KUKA KRL program: EPS_2_251806_MH43A_A_20260213065137.src

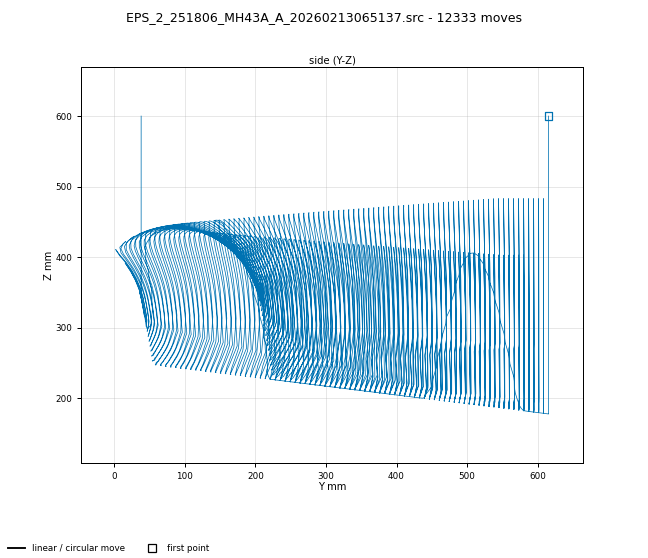
[picture p0: tool path of EPS_2_251806_MH43A_A_20260213065137.src, 12333 of 12335 moves have a stored position in this frame; points joined in program order, loops and branches not executed]
&ACCESS RVP
&REL 4
&COMMENT QRS 19112012
&PARAM EDITMASK = *
DEF PART()
EXT BAS (BAS_COMMAND :IN,REAL :IN )
INT I
BAS (#INITMOV,0 )

;KUKA QRS Post kuka4.cps  Date:22-06-2017 !

File_ID=3028

QRS_PRE_INIT()

;Init var - Until changes are made in qrs_pre_init
Outlet_Square_prg=0
Inlet_1_Square_prg=0
Inlet_2_Square_prg=0
Inlet_3_Square_prg=0
Inlet_4_Square_prg=0
Inlet_5_Square_prg=0

Outlet_1={X 0.000, Y 540.910, Z 382.500, B 0.000, E1 0.000 }
Inlet_1={X 0.000, Y 546.610, Z 302.500, B 0.000, E1 128.000 }
Outlet_1_type=201
Inlet_1_type=201
;QRS#1=Sidecore dimensions
;QRS#2=200-8" PVC SDR 35
;QRS#3=200-8" PVC SDR 35
;QRS#4=
;QRS#5=
;QRS#6=
;QRS#7=
;QRS#8=
;QRS#9=12-08 PSX
;QRS#10=12-08 PSX
;QRS#11=
;QRS#12=
;QRS#13=
;QRS#14=
;QRS#15=
;QRS#16=1220x127x762 2,5'
;QRS#17=EPS Height
;QRS#18=483
;QRS#19=*
;QRS#20= UPDATED VERSION 22-06-2017
;QRS#21=*
Outlet_Square=0100
Inlet_1_Square=0100
Inlet_2_Square=0
Inlet_3_Square=0
Inlet_4_Square=0
Inlet_5_Square=0
Mill_Square=1
Outlet_Square_Prg=204
Inlet_1_Square_prg=204

QRS_INIT()

$ADVANCE=5

; T1
PTP {E1 173.629,E2 173.629}
PTP {X 0,Y 615.469,A -85,B 0,C 180,E1 173.629,E2 173.629,E3 0,E4 0,E5 0,E6 0}
QRS_SPEED_INIT()
LIN {X 0,Y 615.469,Z 600,A -85,B 0,C 180,E1 173.629,E2 173.629,E3 0,E4 0,E5 0,E6 0} C_VEL
LIN {X 0,Y 615.469,Z 187.869,A -85,B 0,C 180,E1 173.629,E2 173.629} C_VEL
LIN {X 0,Y 615.469,Z 179.692,A -85,B 0,C 180,E1 173.629,E2 173.629} C_VEL
LIN {X 0,Y 615.462,Z 177.692,A -85,B 0,C 180,E1 173.442,E2 173.442} C_VEL
LIN {X 0,Y 615.491,Z 177.698,A -85,B 0,C 180,E1 170.801,E2 170.801} C_VEL
LIN {X 0,Y 615.483,Z 177.684,A -85,B 0,C 180,E1 168.139,E2 168.139} C_VEL
LIN {X 0,Y 615.47,Z 177.694,A -85,B 0,C 180,E1 165.451,E2 165.451} C_VEL
LIN {X 0,Y 615.488,Z 177.69,A -85,B 0,C 180,E1 162.73,E2 162.73} C_VEL
LIN {X 0,Y 615.467,Z 177.689,A -85,B 0,C 180,E1 159.967,E2 159.967} C_VEL
LIN {X 0,Y 615.467,Z 177.789,A -85,B 0,C 180,E1 157.786,E2 157.786} C_VEL
LIN {X 0,Y 615.492,Z 192.068,A -85,B 0,C 180,E1 155.008,E2 155.008} C_VEL
LIN {X 0,Y 615.496,Z 193.094,A -85,B 0,C 180,E1 154.81,E2 154.81} C_VEL
LIN {X 0,Y 615.476,Z 299.263,A -85,B 0,C 180,E1 153.537,E2 153.537} C_VEL
LIN {X 0,Y 615.469,Z 311.971,A -85,B 0,C 180,E1 153.256,E2 153.256} C_VEL
LIN {X 0,Y 615.481,Z 325.146,A -85,B 0,C 180,E1 152.822,E2 152.822} C_VEL
LIN {X 0,Y 615.472,Z 337.362,A -85,B 0,C 180,E1 152.269,E2 152.269} C_VEL
LIN {X 0,Y 615.477,Z 348.518,A -85,B 0,C 180,E1 151.617,E2 151.617} C_VEL
LIN {X 0,Y 615.5,Z 358.718,A -85,B 0,C 180,E1 150.876,E2 150.876} C_VEL
LIN {X 0,Y 615.498,Z 368.216,A -85,B 0,C 180,E1 150.022,E2 150.022} C_VEL
LIN {X 0,Y 615.497,Z 376.701,A -85,B 0,C 180,E1 149.081,E2 149.081} C_VEL
LIN {X 0,Y 615.498,Z 383.508,A -85,B 0,C 180,E1 148.154,E2 148.154} C_VEL
LIN {X 0,Y 615.495,Z 389.434,A -85,B 0,C 180,E1 147.154,E2 147.154} C_VEL
LIN {X 0,Y 615.495,Z 394.787,A -85,B 0,C 180,E1 145.978,E2 145.978} C_VEL
LIN {X 0,Y 615.497,Z 398.663,A -85,B 0,C 180,E1 144.786,E2 144.786} C_VEL
LIN {X 0,Y 615.494,Z 401.179,A -85,B 0,C 180,E1 143.576,E2 143.576} C_VEL
LIN {X 0,Y 615.496,Z 402.068,A -85,B 0,C 180,E1 142.758,E2 142.758} C_VEL
LIN {X 0,Y 615.494,Z 402.388,A -85,B 0,C 180,E1 141.932,E2 141.932} C_VEL
LIN {X 0,Y 615.495,Z 401.914,A -85,B 0,C 180,E1 140.937,E2 140.937} C_VEL
LIN {X 0,Y 615.496,Z 400.471,A -85,B 0,C 180,E1 139.91,E2 139.91} C_VEL
LIN {X 0,Y 615.494,Z 398.077,A -85,B 0,C 180,E1 138.905,E2 138.905} C_VEL
LIN {X 0,Y 615.497,Z 394.739,A -85,B 0,C 180,E1 137.919,E2 137.919} C_VEL
LIN {X 0,Y 615.498,Z 389.436,A -85,B 0,C 180,E1 136.756,E2 136.756} C_VEL
LIN {X 0,Y 615.494,Z 382.831,A -85,B 0,C 180,E1 135.656,E2 135.656} C_VEL
LIN {X 0,Y 615.495,Z 375.933,A -85,B 0,C 180,E1 134.735,E2 134.735} C_VEL
LIN {X 0,Y 615.498,Z 367.432,A -85,B 0,C 180,E1 133.808,E2 133.808} C_VEL
LIN {X 0,Y 615.499,Z 357.776,A -85,B 0,C 180,E1 132.961,E2 132.961} C_VEL
LIN {X 0,Y 615.47,Z 347.339,A -85,B 0,C 180,E1 132.216,E2 132.216} C_VEL
LIN {X 0,Y 615.466,Z 337.073,A -85,B 0,C 180,E1 131.625,E2 131.625} C_VEL
LIN {X 0,Y 615.489,Z 325.328,A -85,B 0,C 180,E1 131.094,E2 131.094} C_VEL
LIN {X 0,Y 615.476,Z 312.489,A -85,B 0,C 180,E1 130.668,E2 130.668} C_VEL
LIN {X 0,Y 615.478,Z 299.674,A -85,B 0,C 180,E1 130.381,E2 130.381} C_VEL
LIN {X 0,Y 615.5,Z 193.126,A -85,B 0,C 180,E1 129.106,E2 129.106} C_VEL
LIN {X 0,Y 615.473,Z 179.33,A -85,B 0,C 180,E1 126.426,E2 126.426} C_VEL
LIN {X 0,Y 615.455,Z 177.694,A -85,B 0,C 180,E1 126.09,E2 126.09} C_VEL
LIN {X 0,Y 615.472,Z 177.687,A -85,B 0,C 180,E1 123.532,E2 123.532} C_VEL
LIN {X 0,Y 615.494,Z 177.696,A -85,B 0,C 180,E1 120.919,E2 120.919} C_VEL
LIN {X 0,Y 615.464,Z 177.696,A -85,B 0,C 180,E1 118.446,E2 118.446} C_VEL
LIN {X 0,Y 615.461,Z 177.695,A -85,B 0,C 180,E1 116.445,E2 116.445} C_VEL
LIN {X 0,Y 615.456,Z 177.69,A -85,B 0,C 180,E1 114.001,E2 114.001} C_VEL
LIN {X 0,Y 615.496,Z 177.687,A -85,B 0,C 180,E1 111.431,E2 111.431} C_VEL
LIN {X 0,Y 615.459,Z 177.695,A -85,B 0,C 180,E1 108.596,E2 108.596} C_VEL
LIN {X 0,Y 615.472,Z 177.687,A -85,B 0,C 180,E1 105.905,E2 105.905} C_VEL
LIN {X 0,Y 615.495,Z 177.701,A -85,B 0,C 180,E1 103.201,E2 103.201} C_VEL
LIN {X 0,Y 615.451,Z 177.693,A -85,B 0,C 180,E1 100.527,E2 100.527} C_VEL
LIN {X 0,Y 615.484,Z 177.687,A -85,B 0,C 180,E1 97.875,E2 97.875} C_VEL
LIN {X 0,Y 615.485,Z 177.699,A -85,B 0,C 180,E1 95.241,E2 95.241} C_VEL
LIN {X 0,Y 615.451,Z 177.692,A -85,B 0,C 180,E1 92.618,E2 92.618} C_VEL
LIN {X 0,Y 615.486,Z 177.688,A -85,B 0,C 180,E1 90,E2 90} C_VEL
LIN {X 0,Y 615.48,Z 177.698,A -85,B 0,C 180,E1 87.382,E2 87.382} C_VEL
LIN {X 0,Y 615.447,Z 177.692,A -85,B 0,C 180,E1 84.758,E2 84.758} C_VEL
LIN {X 0,Y 615.489,Z 177.689,A -85,B 0,C 180,E1 82.124,E2 82.124} C_VEL
LIN {X 0,Y 615.47,Z 177.697,A -85,B 0,C 180,E1 79.473,E2 79.473} C_VEL
LIN {X 0,Y 615.455,Z 177.69,A -85,B 0,C 180,E1 76.798,E2 76.798} C_VEL
LIN {X 0,Y 615.495,Z 177.693,A -85,B 0,C 180,E1 74.095,E2 74.095} C_VEL
LIN {X 0,Y 615.451,Z 177.694,A -85,B 0,C 180,E1 71.353,E2 71.353} C_VEL
LIN {X 0,Y 615.448,Z 177.693,A -85,B 0,C 180,E1 69.268,E2 69.268} C_VEL
LIN {X 0,Y 615.488,Z 177.69,A -85,B 0,C 180,E1 66.443,E2 66.443} C_VEL
LIN {X 0,Y 615.45,Z 177.695,A -85,B 0,C 180,E1 63.554,E2 63.554} C_VEL
LIN {X 0,Y 615.448,Z 177.692,A -85,B 0,C 180,E1 61.34,E2 61.34} C_VEL
LIN {X 0,Y 615.474,Z 177.688,A -85,B 0,C 180,E1 58.916,E2 58.916} C_VEL
LIN {X 0,Y 615.465,Z 177.697,A -85,B 0,C 180,E1 55.976,E2 55.976} C_VEL
LIN {X 0,Y 615.445,Z 177.693,A -85,B 0,C 180,E1 53.572,E2 53.572} C_VEL
LIN {X 0,Y 615.491,Z 177.687,A -85,B 0,C 180,E1 50.938,E2 50.938} C_VEL
LIN {X 0,Y 615.495,Z 177.7,A -85,B 0,C 180,E1 48.526,E2 48.526} C_VEL
LIN {X 0,Y 615.446,Z 177.694,A -85,B 0,C 180,E1 45.846,E2 45.846} C_VEL
LIN {X 0,Y 615.488,Z 177.689,A -85,B 0,C 180,E1 43.047,E2 43.047} C_VEL
LIN {X 0,Y 615.481,Z 177.702,A -85,B 0,C 180,E1 40.607,E2 40.607} C_VEL
LIN {X 0,Y 615.444,Z 177.694,A -85,B 0,C 180,E1 38.006,E2 38.006} C_VEL
LIN {X 0,Y 615.454,Z 177.691,A -85,B 0,C 180,E1 35.618,E2 35.618} C_VEL
LIN {X 0,Y 615.488,Z 177.69,A -85,B 0,C 180,E1 33.236,E2 33.236} C_VEL
LIN {X 0,Y 615.493,Z 177.701,A -85,B 0,C 180,E1 30.919,E2 30.919} C_VEL
LIN {X 0,Y 615.451,Z 177.696,A -85,B 0,C 180,E1 28.443,E2 28.443} C_VEL
LIN {X 0,Y 615.449,Z 177.695,A -85,B 0,C 180,E1 26.446,E2 26.446} C_VEL
LIN {X 0,Y 615.449,Z 177.692,A -85,B 0,C 180,E1 23.999,E2 23.999} C_VEL
LIN {X 0,Y 615.497,Z 177.69,A -85,B 0,C 180,E1 21.432,E2 21.432} C_VEL
LIN {X 0,Y 615.444,Z 177.696,A -85,B 0,C 180,E1 18.592,E2 18.592} C_VEL
LIN {X 0,Y 615.443,Z 177.694,A -85,B 0,C 180,E1 16.416,E2 16.416} C_VEL
LIN {X 0,Y 615.477,Z 177.689,A -85,B 0,C 180,E1 13.874,E2 13.874} C_VEL
LIN {X 0,Y 615.476,Z 177.699,A -85,B 0,C 180,E1 11.193,E2 11.193} C_VEL
LIN {X 0,Y 615.442,Z 177.693,A -85,B 0,C 180,E1 8.537,E2 8.537} C_VEL
LIN {X 0,Y 615.496,Z 177.688,A -85,B 0,C 180,E1 5.898,E2 5.898} C_VEL
LIN {X 0,Y 615.466,Z 177.698,A -85,B 0,C 180,E1 3.273,E2 3.273} C_VEL
LIN {X 0,Y 615.465,Z 177.698,A -85,B 0,C 180,E1 1.309,E2 1.309} C_VEL
LIN {X 0,Y 615.442,Z 177.693,A -85,B 0,C 180,E1 -1.309,E2 -1.309} C_VEL
LIN {X 0,Y 615.487,Z 177.692,A -85,B 0,C 180,E1 -3.929,E2 -3.929} C_VEL
LIN {X 0,Y 615.456,Z 177.698,A -85,B 0,C 180,E1 -6.557,E2 -6.557} C_VEL
LIN {X 0,Y 615.458,Z 177.697,A -85,B 0,C 180,E1 -8.537,E2 -8.537} C_VEL
LIN {X 0,Y 615.44,Z 177.695,A -85,B 0,C 180,E1 -10.863,E2 -10.863} C_VEL
LIN {X 0,Y 615.449,Z 177.692,A -85,B 0,C 180,E1 -13.202,E2 -13.202} C_VEL
LIN {X 0,Y 615.493,Z 177.699,A -85,B 0,C 180,E1 -15.905,E2 -15.905} C_VEL
LIN {X 0,Y 615.438,Z 177.696,A -85,B 0,C 180,E1 -18.648,E2 -18.648} C_VEL
LIN {X 0,Y 615.488,Z 177.689,A -85,B 0,C 180,E1 -21.432,E2 -21.432} C_VEL
LIN {X 0,Y 615.449,Z 177.697,A -85,B 0,C 180,E1 -24.274,E2 -24.274} C_VEL
LIN {X 0,Y 615.438,Z 177.696,A -85,B 0,C 180,E1 -26.447,E2 -26.447} C_VEL
LIN {X 0,Y 615.439,Z 177.694,A -85,B 0,C 180,E1 -28.661,E2 -28.661} C_VEL
LIN {X 0,Y 615.471,Z 177.691,A -85,B 0,C 180,E1 -31.083,E2 -31.083} C_VEL
LIN {X 0,Y 615.449,Z 177.697,A -85,B 0,C 180,E1 -34.025,E2 -34.025} C_VEL
LIN {X 0,Y 615.437,Z 177.694,A -85,B 0,C 180,E1 -36.428,E2 -36.428} C_VEL
LIN {X 0,Y 615.49,Z 177.69,A -85,B 0,C 180,E1 -39.062,E2 -39.062} C_VEL
LIN {X 0,Y 615.487,Z 177.699,A -85,B 0,C 180,E1 -41.474,E2 -41.474} C_VEL
LIN {X 0,Y 615.435,Z 177.695,A -85,B 0,C 180,E1 -44.155,E2 -44.155} C_VEL
LIN {X 0,Y 615.473,Z 177.691,A -85,B 0,C 180,E1 -46.754,E2 -46.754} C_VEL
LIN {X 0,Y 615.469,Z 177.7,A -85,B 0,C 180,E1 -49.392,E2 -49.392} C_VEL
LIN {X 0,Y 615.434,Z 177.696,A -85,B 0,C 180,E1 -51.927,E2 -51.927} C_VEL
LIN {X 0,Y 615.449,Z 177.693,A -85,B 0,C 180,E1 -54.381,E2 -54.381} C_VEL
LIN {X 0,Y 615.489,Z 177.694,A -85,B 0,C 180,E1 -56.764,E2 -56.764} C_VEL
LIN {X 0,Y 615.477,Z 177.701,A -85,B 0,C 180,E1 -59.079,E2 -59.079} C_VEL
LIN {X 0,Y 615.437,Z 177.697,A -85,B 0,C 180,E1 -61.559,E2 -61.559} C_VEL
LIN {X 0,Y 615.436,Z 177.696,A -85,B 0,C 180,E1 -63.553,E2 -63.553} C_VEL
LIN {X 0,Y 615.445,Z 177.839,A -85,B 0,C 180,E1 -66.029,E2 -66.029} C_VEL
LIN {X 0,Y 615.472,Z 199.807,A -85,B 0,C 180,E1 -68.743,E2 -68.743} C_VEL
LIN {X 0,Y 615.494,Z 221.654,A -85,B 0,C 180,E1 -71.394,E2 -71.394} C_VEL
LIN {X 0,Y 615.491,Z 245.672,A -85,B 0,C 180,E1 -74.265,E2 -74.265} C_VEL
LIN {X 0,Y 615.455,Z 269.639,A -85,B 0,C 180,E1 -77.092,E2 -77.092} C_VEL
LIN {X 0,Y 615.457,Z 274.667,A -85,B 0,C 180,E1 -77.176,E2 -77.176} C_VEL
LIN {X 0,Y 615.488,Z 378.818,A -85,B 0,C 180,E1 -78.41,E2 -78.41} C_VEL
LIN {X 0,Y 615.477,Z 391.338,A -85,B 0,C 180,E1 -78.681,E2 -78.681} C_VEL
LIN {X 0,Y 615.488,Z 404.617,A -85,B 0,C 180,E1 -79.113,E2 -79.113} C_VEL
LIN {X 0,Y 615.477,Z 416.475,A -85,B 0,C 180,E1 -79.639,E2 -79.639} C_VEL
LIN {X 0,Y 615.494,Z 427.991,A -85,B 0,C 180,E1 -80.304,E2 -80.304} C_VEL
LIN {X 0,Y 615.499,Z 438.338,A -85,B 0,C 180,E1 -81.05,E2 -81.05} C_VEL
LIN {X 0,Y 615.497,Z 446.809,A -85,B 0,C 180,E1 -81.794,E2 -81.794} C_VEL
LIN {X 0,Y 615.498,Z 454.604,A -85,B 0,C 180,E1 -82.619,E2 -82.619} C_VEL
LIN {X 0,Y 615.496,Z 462.202,A -85,B 0,C 180,E1 -83.608,E2 -83.608} C_VEL
LIN {X 0,Y 615.498,Z 469.203,A -85,B 0,C 180,E1 -84.759,E2 -84.759} C_VEL
LIN {X 0,Y 615.494,Z 473.85,A -85,B 0,C 180,E1 -85.743,E2 -85.743} C_VEL
LIN {X 0,Y 615.494,Z 477.398,A -85,B 0,C 180,E1 -86.727,E2 -86.727} C_VEL
LIN {X 0,Y 615.497,Z 479.232,A -85,B 0,C 180,E1 -87.382,E2 -87.382} C_VEL
LIN {X 0,Y 615.5,Z 480.607,A -85,B 0,C 180,E1 -88.037,E2 -88.037} C_VEL
LIN {X 0,Y 615.496,Z 482.173,A -85,B 0,C 180,E1 -89.346,E2 -89.346} C_VEL
LIN {X 0,Y 615.494,Z 482.389,A -85,B 0,C 180,E1 -90,E2 -90} C_VEL
LIN {X 0,Y 615.495,Z 481.58,A -85,B 0,C 180,E1 -91.308,E2 -91.308} C_VEL
LIN {X 0,Y 615.5,Z 480.608,A -85,B 0,C 180,E1 -91.963,E2 -91.963} C_VEL
LIN {X 0,Y 615.497,Z 479.233,A -85,B 0,C 180,E1 -92.618,E2 -92.618} C_VEL
LIN {X 0,Y 615.496,Z 476.35,A -85,B 0,C 180,E1 -93.6,E2 -93.6} C_VEL
LIN {X 0,Y 615.498,Z 472.442,A -85,B 0,C 180,E1 -94.584,E2 -94.584} C_VEL
LIN {X 0,Y 615.499,Z 467.406,A -85,B 0,C 180,E1 -95.57,E2 -95.57} C_VEL
LIN {X 0,Y 615.497,Z 460.87,A -85,B 0,C 180,E1 -96.583,E2 -96.583} C_VEL
LIN {X 0,Y 615.497,Z 453.134,A -85,B 0,C 180,E1 -97.545,E2 -97.545} C_VEL
LIN {X 0,Y 615.498,Z 445.047,A -85,B 0,C 180,E1 -98.371,E2 -98.371} C_VEL
LIN {X 0,Y 615.499,Z 435.169,A -85,B 0,C 180,E1 -99.198,E2 -99.198} C_VEL
LIN {X 0,Y 615.488,Z 423.984,A -85,B 0,C 180,E1 -99.945,E2 -99.945} C_VEL
LIN {X 0,Y 615.482,Z 413.027,A -85,B 0,C 180,E1 -100.527,E2 -100.527} C_VEL
LIN {X 0,Y 615.48,Z 400.492,A -85,B 0,C 180,E1 -101.04,E2 -101.04} C_VEL
LIN {X 0,Y 615.479,Z 388.073,A -85,B 0,C 180,E1 -101.402,E2 -101.402} C_VEL
LIN {X 0,Y 615.493,Z 374.475,A -85,B 0,C 180,E1 -101.652,E2 -101.652} C_VEL
LIN {X 0,Y 615.455,Z 269.821,A -85,B 0,C 180,E1 -102.887,E2 -102.887} C_VEL
LIN {X 0,Y 615.493,Z 247.108,A -85,B 0,C 180,E1 -105.565,E2 -105.565} C_VEL
LIN {X 0,Y 615.49,Z 223.006,A -85,B 0,C 180,E1 -108.443,E2 -108.443} C_VEL
LIN {X 0,Y 615.46,Z 201.245,A -85,B 0,C 180,E1 -111.082,E2 -111.082} C_VEL
LIN {X 0,Y 615.447,Z 178.059,A -85,B 0,C 180,E1 -113.943,E2 -113.943} C_VEL
LIN {X 0,Y 615.443,Z 177.694,A -85,B 0,C 180,E1 -113.999,E2 -113.999} C_VEL
LIN {X 0,Y 615.437,Z 177.696,A -85,B 0,C 180,E1 -116.446,E2 -116.446} C_VEL
LIN {X 0,Y 615.485,Z 177.692,A -85,B 0,C 180,E1 -119.406,E2 -119.406} C_VEL
LIN {X 0,Y 615.455,Z 177.692,A -85,B 0,C 180,E1 -121.687,E2 -121.687} C_VEL
LIN {X 0,Y 615.438,Z 177.694,A -85,B 0,C 180,E1 -124.025,E2 -124.025} C_VEL
LIN {X 0,Y 615.489,Z 177.699,A -85,B 0,C 180,E1 -126.936,E2 -126.936} C_VEL
LIN {X 0,Y 615.441,Z 177.693,A -85,B 0,C 180,E1 -129.754,E2 -129.754} C_VEL
LIN {X 0,Y 615.462,Z 177.698,A -85,B 0,C 180,E1 -132.355,E2 -132.355} C_VEL
LIN {X 0,Y 615.491,Z 177.688,A -85,B 0,C 180,E1 -135.068,E2 -135.068} C_VEL
LIN {X 0,Y 615.444,Z 177.693,A -85,B 0,C 180,E1 -137.643,E2 -137.643} C_VEL
LIN {X 0,Y 615.474,Z 177.698,A -85,B 0,C 180,E1 -140.249,E2 -140.249} C_VEL
LIN {X 0,Y 615.471,Z 177.689,A -85,B 0,C 180,E1 -143.065,E2 -143.065} C_VEL
LIN {X 0,Y 615.452,Z 177.691,A -85,B 0,C 180,E1 -145.304,E2 -145.304} C_VEL
LIN {X 0,Y 615.451,Z 177.695,A -85,B 0,C 180,E1 -147.675,E2 -147.675} C_VEL
LIN {X 0,Y 615.499,Z 177.7,A -85,B 0,C 180,E1 -150.203,E2 -150.203} C_VEL
LIN {X 0,Y 615.462,Z 177.689,A -85,B 0,C 180,E1 -152.96,E2 -152.96} C_VEL
LIN {X 0,Y 615.458,Z 177.69,A -85,B 0,C 180,E1 -155.007,E2 -155.007} C_VEL
LIN {X 0,Y 615.467,Z 177.697,A -85,B 0,C 180,E1 -157.659,E2 -157.659} C_VEL
LIN {X 0,Y 615.475,Z 177.687,A -85,B 0,C 180,E1 -160.662,E2 -160.662} C_VEL
LIN {X 0,Y 615.466,Z 177.688,A -85,B 0,C 180,E1 -162.729,E2 -162.729} C_VEL
LIN {X 0,Y 615.469,Z 177.697,A -85,B 0,C 180,E1 -165.45,E2 -165.45} C_VEL
LIN {X 0,Y 615.488,Z 177.689,A -85,B 0,C 180,E1 -168.139,E2 -168.139} C_VEL
LIN {X 0,Y 615.457,Z 177.69,A -85,B 0,C 180,E1 -170.801,E2 -170.801} C_VEL
LIN {X 0,Y 615.49,Z 177.699,A -85,B 0,C 180,E1 -173.443,E2 -173.443} C_VEL
LIN {X 0,Y 615.487,Z 177.686,A -85,B 0,C 180,E1 -176.071,E2 -176.071} C_VEL
LIN {X 0,Y 615.459,Z 177.691,A -85,B 0,C 180,E1 -178.691,E2 -178.691} C_VEL
LIN {X 0,Y 615.492,Z 177.702,A -85,B 0,C 180,E1 -181.309,E2 -181.309} C_VEL
LIN {X 0,Y 615.486,Z 177.685,A -85,B 0,C 180,E1 -183.928,E2 -183.928} C_VEL
LIN {X 0,Y 615.462,Z 177.692,A -85,B 0,C 180,E1 -186.558,E2 -186.558} C_VEL
LIN {X 0,Y 614.804,Z 177.845,A -85,B 0,C 180,E1 -187.104,E2 -187.104} C_VEL
LIN {X 0,Y 611.985,Z 178.248,A -85,B 0,C 180,E1 -187.99,E2 -187.99} C_VEL
LIN {X 0,Y 609.595,Z 178.562,A -85,B 0,C 180,E1 -188.703,E2 -188.703} C_VEL
LIN {X 0,Y 608.556,Z 178.683,A -85,B 0,C 180,E1 -189.252,E2 -189.252} C_VEL
LIN {X 0,Y 608.464,Z 178.691,A -85,B 0,C 180,E1 -189.438,E2 -189.438} C_VEL
LIN {X 0,Y 608.456,Z 178.687,A -85,B 0,C 180,E1 -192,E2 -192} C_VEL
LIN {X 0,Y 608.466,Z 178.693,A -85,B 0,C 180,E1 -194.721,E2 -194.721} C_VEL
LIN {X 0,Y 608.45,Z 178.69,A -85,B 0,C 180,E1 -197.477,E2 -197.477} C_VEL
LIN {X 0,Y 608.449,Z 178.691,A -85,B 0,C 180,E1 -200.275,E2 -200.275} C_VEL
LIN {X 0,Y 608.454,Z 178.73,A -85,B 0,C 180,E1 -202.183,E2 -202.183} C_VEL
LIN {X 0,Y 608.474,Z 192.782,A -85,B 0,C 180,E1 -204.935,E2 -204.935} C_VEL
LIN {X 0,Y 608.458,Z 193.373,A -85,B 0,C 180,E1 -205.049,E2 -205.049} C_VEL
LIN {X 0,Y 608.535,Z 299.465,A -85,B 0,C 180,E1 -206.331,E2 -206.331} C_VEL
LIN {X 0,Y 608.52,Z 312.77,A -85,B 0,C 180,E1 -206.632,E2 -206.632} C_VEL
LIN {X 0,Y 608.504,Z 323.878,A -85,B 0,C 180,E1 -206.999,E2 -206.999} C_VEL
LIN {X 0,Y 608.502,Z 335.659,A -85,B 0,C 180,E1 -207.515,E2 -207.515} C_VEL
LIN {X 0,Y 608.458,Z 347.236,A -85,B 0,C 180,E1 -208.173,E2 -208.173} C_VEL
LIN {X 0,Y 608.486,Z 357.461,A -85,B 0,C 180,E1 -208.901,E2 -208.901} C_VEL
LIN {X 0,Y 608.483,Z 367.48,A -85,B 0,C 180,E1 -209.779,E2 -209.779} C_VEL
LIN {X 0,Y 608.459,Z 376.171,A -85,B 0,C 180,E1 -210.726,E2 -210.726} C_VEL
LIN {X 0,Y 608.463,Z 383.466,A -85,B 0,C 180,E1 -211.705,E2 -211.705} C_VEL
LIN {X 0,Y 608.432,Z 388.454,A -85,B 0,C 180,E1 -212.518,E2 -212.518} C_VEL
LIN {X 0,Y 608.425,Z 394.325,A -85,B 0,C 180,E1 -213.728,E2 -213.728} C_VEL
LIN {X 0,Y 608.427,Z 398.485,A -85,B 0,C 180,E1 -214.903,E2 -214.903} C_VEL
LIN {X 0,Y 608.422,Z 401.259,A -85,B 0,C 180,E1 -216.094,E2 -216.094} C_VEL
LIN {X 0,Y 608.435,Z 402.622,A -85,B 0,C 180,E1 -217.154,E2 -217.154} C_VEL
LIN {X 0,Y 608.42,Z 402.962,A -85,B 0,C 180,E1 -218.235,E2 -218.235} C_VEL
LIN {X 0,Y 608.423,Z 402.096,A -85,B 0,C 180,E1 -219.443,E2 -219.443} C_VEL
LIN {X 0,Y 608.433,Z 399.686,A -85,B 0,C 180,E1 -220.74,E2 -220.74} C_VEL
LIN {X 0,Y 608.45,Z 396.943,A -85,B 0,C 180,E1 -221.673,E2 -221.673} C_VEL
LIN {X 0,Y 608.442,Z 393.221,A -85,B 0,C 180,E1 -222.62,E2 -222.62} C_VEL
LIN {X 0,Y 608.453,Z 388.509,A -85,B 0,C 180,E1 -223.562,E2 -223.562} C_VEL
LIN {X 0,Y 608.459,Z 381.684,A -85,B 0,C 180,E1 -224.648,E2 -224.648} C_VEL
LIN {X 0,Y 608.469,Z 372.97,A -85,B 0,C 180,E1 -225.735,E2 -225.735} C_VEL
LIN {X 0,Y 608.476,Z 364.473,A -85,B 0,C 180,E1 -226.595,E2 -226.595} C_VEL
LIN {X 0,Y 608.478,Z 354.93,A -85,B 0,C 180,E1 -227.386,E2 -227.386} C_VEL
LIN {X 0,Y 608.475,Z 343.681,A -85,B 0,C 180,E1 -228.135,E2 -228.135} C_VEL
LIN {X 0,Y 608.512,Z 331.514,A -85,B 0,C 180,E1 -228.774,E2 -228.774} C_VEL
LIN {X 0,Y 608.526,Z 318.947,A -85,B 0,C 180,E1 -229.268,E2 -229.268} C_VEL
LIN {X 0,Y 608.518,Z 305.883,A -85,B 0,C 180,E1 -229.632,E2 -229.632} C_VEL
LIN {X 0,Y 608.543,Z 293.08,A -85,B 0,C 180,E1 -229.853,E2 -229.853} C_VEL
LIN {X 0,Y 608.5,Z 193.71,A -85,B 0,C 180,E1 -231.03,E2 -231.03} C_VEL
LIN {X 0,Y 608.473,Z 193.319,A -85,B 0,C 180,E1 -231.051,E2 -231.051} C_VEL
LIN {X 0,Y 608.458,Z 179.763,A -85,B 0,C 180,E1 -233.704,E2 -233.704} C_VEL
LIN {X 0,Y 608.437,Z 178.692,A -85,B 0,C 180,E1 -233.956,E2 -233.956} C_VEL
LIN {X 0,Y 608.443,Z 178.689,A -85,B 0,C 180,E1 -236.328,E2 -236.328} C_VEL
LIN {X 0,Y 608.449,Z 178.691,A -85,B 0,C 180,E1 -238.732,E2 -238.732} C_VEL
LIN {X 0,Y 608.463,Z 178.693,A -85,B 0,C 180,E1 -241.382,E2 -241.382} C_VEL
LIN {X 0,Y 608.427,Z 178.691,A -85,B 0,C 180,E1 -243.964,E2 -243.964} C_VEL
LIN {X 0,Y 608.447,Z 178.688,A -85,B 0,C 180,E1 -246.154,E2 -246.154} C_VEL
LIN {X 0,Y 608.453,Z 178.698,A -85,B 0,C 180,E1 -249.019,E2 -249.019} C_VEL
LIN {X 0,Y 608.426,Z 178.691,A -85,B 0,C 180,E1 -251.828,E2 -251.828} C_VEL
LIN {X 0,Y 608.474,Z 178.691,A -85,B 0,C 180,E1 -254.594,E2 -254.594} C_VEL
LIN {X 0,Y 608.453,Z 178.69,A -85,B 0,C 180,E1 -257.323,E2 -257.323} C_VEL
LIN {X 0,Y 608.453,Z 178.688,A -85,B 0,C 180,E1 -260.023,E2 -260.023} C_VEL
LIN {X 0,Y 608.461,Z 178.697,A -85,B 0,C 180,E1 -262.701,E2 -262.701} C_VEL
LIN {X 0,Y 608.465,Z 178.695,A -85,B 0,C 180,E1 -264.698,E2 -264.698} C_VEL
LIN {X 0,Y 608.447,Z 178.689,A -85,B 0,C 180,E1 -267.352,E2 -267.352} C_VEL
LIN {X 0,Y 608.477,Z 178.687,A -85,B 0,C 180,E1 -270,E2 -270} C_VEL
LIN {X 0,Y 608.47,Z 178.692,A -85,B 0,C 180,E1 -272.648,E2 -272.648} C_VEL
LIN {X 0,Y 608.433,Z 178.69,A -85,B 0,C 180,E1 -275.302,E2 -275.302} C_VEL
LIN {X 0,Y 608.478,Z 178.689,A -85,B 0,C 180,E1 -277.967,E2 -277.967} C_VEL
LIN {X 0,Y 608.443,Z 178.693,A -85,B 0,C 180,E1 -280.65,E2 -280.65} C_VEL
LIN {X 0,Y 608.444,Z 178.689,A -85,B 0,C 180,E1 -283.357,E2 -283.357} C_VEL
LIN {X 0,Y 608.459,Z 178.697,A -85,B 0,C 180,E1 -286.094,E2 -286.094} C_VEL
LIN {X 0,Y 608.44,Z 178.689,A -85,B 0,C 180,E1 -288.87,E2 -288.87} C_VEL
LIN {X 0,Y 608.469,Z 178.691,A -85,B 0,C 180,E1 -291.692,E2 -291.692} C_VEL
LIN {X 0,Y 608.432,Z 178.691,A -85,B 0,C 180,E1 -294.572,E2 -294.572} C_VEL
LIN {X 0,Y 608.466,Z 178.687,A -85,B 0,C 180,E1 -297.205,E2 -297.205} C_VEL
LIN {X 0,Y 608.45,Z 178.695,A -85,B 0,C 180,E1 -299.968,E2 -299.968} C_VEL
LIN {X 0,Y 608.444,Z 178.689,A -85,B 0,C 180,E1 -302.881,E2 -302.881} C_VEL
LIN {X 0,Y 608.44,Z 178.693,A -85,B 0,C 180,E1 -305.278,E2 -305.278} C_VEL
LIN {X 0,Y 608.456,Z 178.695,A -85,B 0,C 180,E1 -307.748,E2 -307.748} C_VEL
LIN {X 0,Y 608.435,Z 178.69,A -85,B 0,C 180,E1 -310.327,E2 -310.327} C_VEL
LIN {X 0,Y 608.449,Z 178.69,A -85,B 0,C 180,E1 -312.961,E2 -312.961} C_VEL
LIN {X 0,Y 608.433,Z 178.695,A -85,B 0,C 180,E1 -315.739,E2 -315.739} C_VEL
LIN {X 0,Y 608.433,Z 178.692,A -85,B 0,C 180,E1 -317.936,E2 -317.936} C_VEL
LIN {X 0,Y 608.442,Z 178.691,A -85,B 0,C 180,E1 -320.706,E2 -320.706} C_VEL
LIN {X 0,Y 608.457,Z 178.695,A -85,B 0,C 180,E1 -323.085,E2 -323.085} C_VEL
LIN {X 0,Y 608.458,Z 178.691,A -85,B 0,C 180,E1 -325.53,E2 -325.53} C_VEL
LIN {X 0,Y 608.436,Z 178.69,A -85,B 0,C 180,E1 -327.904,E2 -327.904} C_VEL
LIN {X 0,Y 608.441,Z 178.689,A -85,B 0,C 180,E1 -330.219,E2 -330.219} C_VEL
LIN {X 0,Y 608.488,Z 178.69,A -85,B 0,C 180,E1 -332.792,E2 -332.792} C_VEL
LIN {X 0,Y 608.435,Z 178.693,A -85,B 0,C 180,E1 -335.428,E2 -335.428} C_VEL
LIN {X 0,Y 608.461,Z 178.688,A -85,B 0,C 180,E1 -338.308,E2 -338.308} C_VEL
LIN {X 0,Y 608.426,Z 178.694,A -85,B 0,C 180,E1 -341.297,E2 -341.297} C_VEL
LIN {X 0,Y 608.436,Z 178.69,A -85,B 0,C 180,E1 -343.906,E2 -343.906} C_VEL
LIN {X 0,Y 608.461,Z 178.697,A -85,B 0,C 180,E1 -346.644,E2 -346.644} C_VEL
LIN {X 0,Y 608.425,Z 178.692,A -85,B 0,C 180,E1 -349.349,E2 -349.349} C_VEL
LIN {X 0,Y 608.471,Z 178.688,A -85,B 0,C 180,E1 -352.033,E2 -352.033} C_VEL
LIN {X 0,Y 608.451,Z 178.695,A -85,B 0,C 180,E1 -354.698,E2 -354.698} C_VEL
LIN {X 0,Y 608.439,Z 178.689,A -85,B 0,C 180,E1 -357.352,E2 -357.352} C_VEL
LIN {X 0,Y 608.477,Z 178.689,A -85,B 0,C 180,E1 -360,E2 -360} C_VEL
LIN {X 0,Y 608.455,Z 178.692,A -85,B 0,C 180,E1 -362.648,E2 -362.648} C_VEL
LIN {X 0,Y 608.428,Z 178.691,A -85,B 0,C 180,E1 -365.302,E2 -365.302} C_VEL
LIN {X 0,Y 608.477,Z 178.691,A -85,B 0,C 180,E1 -367.967,E2 -367.967} C_VEL
LIN {X 0,Y 608.43,Z 178.693,A -85,B 0,C 180,E1 -370.651,E2 -370.651} C_VEL
LIN {X 0,Y 608.44,Z 178.69,A -85,B 0,C 180,E1 -373.357,E2 -373.357} C_VEL
LIN {X 0,Y 608.453,Z 178.696,A -85,B 0,C 180,E1 -376.094,E2 -376.094} C_VEL
LIN {X 0,Y 608.435,Z 178.69,A -85,B 0,C 180,E1 -378.87,E2 -378.87} C_VEL
LIN {X 0,Y 608.462,Z 178.694,A -85,B 0,C 180,E1 -381.692,E2 -381.692} C_VEL
LIN {X 0,Y 608.423,Z 178.692,A -85,B 0,C 180,E1 -384.572,E2 -384.572} C_VEL
LIN {X 0,Y 608.464,Z 178.689,A -85,B 0,C 180,E1 -387.204,E2 -387.204} C_VEL
LIN {X 0,Y 608.435,Z 178.695,A -85,B 0,C 180,E1 -389.966,E2 -389.966} C_VEL
LIN {X 0,Y 608.421,Z 178.691,A -85,B 0,C 180,E1 -392.516,E2 -392.516} C_VEL
LIN {X 0,Y 608.432,Z 178.696,A -85,B 0,C 180,E1 -395.279,E2 -395.279} C_VEL
LIN {X 0,Y 608.447,Z 178.694,A -85,B 0,C 180,E1 -397.748,E2 -397.748} C_VEL
LIN {X 0,Y 608.436,Z 178.69,A -85,B 0,C 180,E1 -400.327,E2 -400.327} C_VEL
LIN {X 0,Y 608.482,Z 178.694,A -85,B 0,C 180,E1 -403.31,E2 -403.31} C_VEL
LIN {X 0,Y 608.431,Z 178.69,A -85,B 0,C 180,E1 -406.127,E2 -406.127} C_VEL
LIN {X 0,Y 608.448,Z 178.692,A -85,B 0,C 180,E1 -408.823,E2 -408.823} C_VEL
LIN {X 0,Y 608.432,Z 178.692,A -85,B 0,C 180,E1 -411.764,E2 -411.764} C_VEL
LIN {X 0,Y 608.43,Z 178.69,A -85,B 0,C 180,E1 -413.957,E2 -413.957} C_VEL
LIN {X 0,Y 608.446,Z 178.689,A -85,B 0,C 180,E1 -416.328,E2 -416.328} C_VEL
LIN {X 0,Y 608.446,Z 178.695,A -85,B 0,C 180,E1 -418.733,E2 -418.733} C_VEL
LIN {X 0,Y 608.438,Z 178.692,A -85,B 0,C 180,E1 -421.387,E2 -421.387} C_VEL
LIN {X 0,Y 608.427,Z 178.695,A -85,B 0,C 180,E1 -423.224,E2 -423.224} C_VEL
LIN {X 0,Y 608.441,Z 178.789,A -85,B 0,C 180,E1 -425.856,E2 -425.856} C_VEL
LIN {X 0,Y 608.571,Z 189.764,A -85,B 0,C 180,E1 -427.24,E2 -427.24} C_VEL
LIN {X 0,Y 608.572,Z 211.287,A -85,B 0,C 180,E1 -429.906,E2 -429.906} C_VEL
LIN {X 0,Y 608.536,Z 232.812,A -85,B 0,C 180,E1 -432.526,E2 -432.526} C_VEL
LIN {X 0,Y 608.464,Z 254.338,A -85,B 0,C 180,E1 -435.108,E2 -435.108} C_VEL
LIN {X 0,Y 608.488,Z 270.229,A -85,B 0,C 180,E1 -436.973,E2 -436.973} C_VEL
LIN {X 0,Y 608.546,Z 378.935,A -85,B 0,C 180,E1 -438.276,E2 -438.276} C_VEL
LIN {X 0,Y 608.512,Z 392.209,A -85,B 0,C 180,E1 -438.571,E2 -438.571} C_VEL
LIN {X 0,Y 608.514,Z 404.627,A -85,B 0,C 180,E1 -438.982,E2 -438.982} C_VEL
LIN {X 0,Y 608.499,Z 416.631,A -85,B 0,C 180,E1 -439.519,E2 -439.519} C_VEL
LIN {X 0,Y 608.484,Z 428.194,A -85,B 0,C 180,E1 -440.191,E2 -440.191} C_VEL
LIN {X 0,Y 608.485,Z 438.591,A -85,B 0,C 180,E1 -440.946,E2 -440.946} C_VEL
LIN {X 0,Y 608.475,Z 447.11,A -85,B 0,C 180,E1 -441.699,E2 -441.699} C_VEL
LIN {X 0,Y 608.471,Z 454.959,A -85,B 0,C 180,E1 -442.534,E2 -442.534} C_VEL
LIN {X 0,Y 608.461,Z 462.286,A -85,B 0,C 180,E1 -443.484,E2 -443.484} C_VEL
LIN {X 0,Y 608.451,Z 467.865,A -85,B 0,C 180,E1 -444.365,E2 -444.365} C_VEL
LIN {X 0,Y 608.432,Z 472.949,A -85,B 0,C 180,E1 -445.362,E2 -445.362} C_VEL
LIN {X 0,Y 608.449,Z 476.896,A -85,B 0,C 180,E1 -446.357,E2 -446.357} C_VEL
LIN {X 0,Y 608.425,Z 479.809,A -85,B 0,C 180,E1 -447.352,E2 -447.352} C_VEL
LIN {X 0,Y 608.445,Z 481.201,A -85,B 0,C 180,E1 -448.014,E2 -448.014} C_VEL
LIN {X 0,Y 608.439,Z 482.783,A -85,B 0,C 180,E1 -449.338,E2 -449.338} C_VEL
LIN {X 0,Y 608.434,Z 483,A -85,B 0,C 180,E1 -450,E2 -450} C_VEL
LIN {X 0,Y 608.448,Z 482.184,A -85,B 0,C 180,E1 -451.324,E2 -451.324} C_VEL
LIN {X 0,Y 608.445,Z 481.202,A -85,B 0,C 180,E1 -451.986,E2 -451.986} C_VEL
LIN {X 0,Y 608.425,Z 479.81,A -85,B 0,C 180,E1 -452.648,E2 -452.648} C_VEL
LIN {X 0,Y 608.449,Z 476.897,A -85,B 0,C 180,E1 -453.642,E2 -453.642} C_VEL
LIN {X 0,Y 608.432,Z 472.951,A -85,B 0,C 180,E1 -454.638,E2 -454.638} C_VEL
LIN {X 0,Y 608.438,Z 466.878,A -85,B 0,C 180,E1 -455.801,E2 -455.801} C_VEL
LIN {X 0,Y 608.462,Z 460.236,A -85,B 0,C 180,E1 -456.799,E2 -456.799} C_VEL
LIN {X 0,Y 608.456,Z 451.991,A -85,B 0,C 180,E1 -457.8,E2 -457.8} C_VEL
LIN {X 0,Y 608.472,Z 443.538,A -85,B 0,C 180,E1 -458.636,E2 -458.636} C_VEL
LIN {X 0,Y 608.479,Z 433.093,A -85,B 0,C 180,E1 -459.473,E2 -459.473} C_VEL
LIN {X 0,Y 608.489,Z 422.759,A -85,B 0,C 180,E1 -460.145,E2 -460.145} C_VEL
LIN {X 0,Y 608.519,Z 411.269,A -85,B 0,C 180,E1 -460.74,E2 -460.74} C_VEL
LIN {X 0,Y 608.528,Z 398.894,A -85,B 0,C 180,E1 -461.225,E2 -461.225} C_VEL
LIN {X 0,Y 608.544,Z 385.445,A -85,B 0,C 180,E1 -461.597,E2 -461.597} C_VEL
LIN {X 0,Y 608.55,Z 373.096,A -85,B 0,C 180,E1 -461.808,E2 -461.808} C_VEL
LIN {X 0,Y 608.457,Z 269.947,A -85,B 0,C 180,E1 -463.038,E2 -463.038} C_VEL
LIN {X 0,Y 608.515,Z 245.731,A -85,B 0,C 180,E1 -465.92,E2 -465.92} C_VEL
LIN {X 0,Y 608.566,Z 222.355,A -85,B 0,C 180,E1 -468.742,E2 -468.742} C_VEL
LIN {X 0,Y 608.591,Z 199.81,A -85,B 0,C 180,E1 -471.509,E2 -471.509} C_VEL
LIN {X 0,Y 608.56,Z 179.443,A -85,B 0,C 180,E1 -474.057,E2 -474.057} C_VEL
LIN {X 0,Y 608.427,Z 178.693,A -85,B 0,C 180,E1 -474.189,E2 -474.189} C_VEL
LIN {X 0,Y 608.429,Z 178.695,A -85,B 0,C 180,E1 -476.775,E2 -476.775} C_VEL
LIN {X 0,Y 608.428,Z 178.701,A -85,B 0,C 180,E1 -479.022,E2 -479.022} C_VEL
LIN {X 0,Y 608.443,Z 178.694,A -85,B 0,C 180,E1 -481.318,E2 -481.318} C_VEL
LIN {X 0,Y 608.425,Z 178.692,A -85,B 0,C 180,E1 -483.728,E2 -483.728} C_VEL
LIN {X 0,Y 608.431,Z 178.691,A -85,B 0,C 180,E1 -486.093,E2 -486.093} C_VEL
LIN {X 0,Y 608.429,Z 178.697,A -85,B 0,C 180,E1 -488.591,E2 -488.591} C_VEL
LIN {X 0,Y 608.447,Z 178.69,A -85,B 0,C 180,E1 -491.34,E2 -491.34} C_VEL
LIN {X 0,Y 608.437,Z 178.69,A -85,B 0,C 180,E1 -493.872,E2 -493.872} C_VEL
LIN {X 0,Y 608.481,Z 178.692,A -85,B 0,C 180,E1 -496.69,E2 -496.69} C_VEL
LIN {X 0,Y 608.459,Z 178.692,A -85,B 0,C 180,E1 -498.823,E2 -498.823} C_VEL
LIN {X 0,Y 608.443,Z 178.69,A -85,B 0,C 180,E1 -501.763,E2 -501.763} C_VEL
LIN {X 0,Y 608.44,Z 178.693,A -85,B 0,C 180,E1 -503.955,E2 -503.955} C_VEL
LIN {X 0,Y 608.463,Z 178.696,A -85,B 0,C 180,E1 -506.329,E2 -506.329} C_VEL
LIN {X 0,Y 608.445,Z 178.691,A -85,B 0,C 180,E1 -508.733,E2 -508.733} C_VEL
LIN {X 0,Y 608.443,Z 178.689,A -85,B 0,C 180,E1 -511.385,E2 -511.385} C_VEL
LIN {X 0,Y 608.436,Z 178.698,A -85,B 0,C 180,E1 -513.964,E2 -513.964} C_VEL
LIN {X 0,Y 608.434,Z 178.69,A -85,B 0,C 180,E1 -516.875,E2 -516.875} C_VEL
LIN {X 0,Y 608.444,Z 178.69,A -85,B 0,C 180,E1 -519.327,E2 -519.327} C_VEL
LIN {X 0,Y 608.444,Z 178.699,A -85,B 0,C 180,E1 -521.828,E2 -521.828} C_VEL
LIN {X 0,Y 608.456,Z 178.687,A -85,B 0,C 180,E1 -524.594,E2 -524.594} C_VEL
LIN {X 0,Y 608.462,Z 178.691,A -85,B 0,C 180,E1 -527.323,E2 -527.323} C_VEL
LIN {X 0,Y 608.463,Z 178.69,A -85,B 0,C 180,E1 -530.023,E2 -530.023} C_VEL
LIN {X 0,Y 608.431,Z 178.691,A -85,B 0,C 180,E1 -532.7,E2 -532.7} C_VEL
LIN {X 0,Y 608.441,Z 178.689,A -85,B 0,C 180,E1 -534.698,E2 -534.698} C_VEL
LIN {X 0,Y 608.482,Z 178.693,A -85,B 0,C 180,E1 -537.352,E2 -537.352} C_VEL
LIN {X 0,Y 608.477,Z 178.686,A -85,B 0,C 180,E1 -540,E2 -540} C_VEL
LIN {X 0,Y 608.455,Z 178.689,A -85,B 0,C 180,E1 -542.648,E2 -542.648} C_VEL
LIN {X 0,Y 608.472,Z 178.694,A -85,B 0,C 180,E1 -545.302,E2 -545.302} C_VEL
LIN {X 0,Y 608.474,Z 178.685,A -85,B 0,C 180,E1 -547.967,E2 -547.967} C_VEL
LIN {X 0,Y 608.464,Z 178.691,A -85,B 0,C 180,E1 -549.438,E2 -549.438} C_VEL
LIN {X 0,Y 607.78,Z 178.774,A -85,B 0,C 180,E1 -549.991,E2 -549.991} C_VEL
LIN {X 0,Y 604.924,Z 179.135,A -85,B 0,C 180,E1 -550.888,E2 -550.888} C_VEL
LIN {X 0,Y 602.52,Z 179.43,A -85,B 0,C 180,E1 -551.609,E2 -551.609} C_VEL
LIN {X 0,Y 601.488,Z 179.556,A -85,B 0,C 180,E1 -552.166,E2 -552.166} C_VEL
LIN {X 0,Y 601.403,Z 179.568,A -85,B 0,C 180,E1 -552.354,E2 -552.354} C_VEL
LIN {X 0,Y 601.424,Z 179.574,A -85,B 0,C 180,E1 -554.897,E2 -554.897} C_VEL
LIN {X 0,Y 601.391,Z 179.568,A -85,B 0,C 180,E1 -557.689,E2 -557.689} C_VEL
LIN {X 0,Y 601.424,Z 179.57,A -85,B 0,C 180,E1 -560.522,E2 -560.522} C_VEL
LIN {X 0,Y 601.411,Z 179.677,A -85,B 0,C 180,E1 -562.181,E2 -562.181} C_VEL
LIN {X 0,Y 601.425,Z 193.416,A -85,B 0,C 180,E1 -564.901,E2 -564.901} C_VEL
LIN {X 0,Y 601.658,Z 201.73,A -85,B 0,C 180,E1 -565.006,E2 -565.006} C_VEL
LIN {X 0,Y 601.599,Z 299.082,A -85,B 0,C 180,E1 -566.187,E2 -566.187} C_VEL
LIN {X 0,Y 601.553,Z 311.896,A -85,B 0,C 180,E1 -566.473,E2 -566.473} C_VEL
LIN {X 0,Y 601.547,Z 323.939,A -85,B 0,C 180,E1 -566.872,E2 -566.872} C_VEL
LIN {X 0,Y 601.508,Z 336.491,A -85,B 0,C 180,E1 -567.433,E2 -567.433} C_VEL
LIN {X 0,Y 601.449,Z 347.225,A -85,B 0,C 180,E1 -568.055,E2 -568.055} C_VEL
LIN {X 0,Y 601.452,Z 358.495,A -85,B 0,C 180,E1 -568.876,E2 -568.876} C_VEL
LIN {X 0,Y 601.413,Z 368.438,A -85,B 0,C 180,E1 -569.778,E2 -569.778} C_VEL
LIN {X 0,Y 601.407,Z 377.043,A -85,B 0,C 180,E1 -570.748,E2 -570.748} C_VEL
LIN {X 0,Y 601.395,Z 384.114,A -85,B 0,C 180,E1 -571.727,E2 -571.727} C_VEL
LIN {X 0,Y 601.367,Z 389.825,A -85,B 0,C 180,E1 -572.707,E2 -572.707} C_VEL
LIN {X 0,Y 601.363,Z 394.076,A -85,B 0,C 180,E1 -573.619,E2 -573.619} C_VEL
LIN {X 0,Y 601.341,Z 398.679,A -85,B 0,C 180,E1 -574.937,E2 -574.937} C_VEL
LIN {X 0,Y 601.315,Z 401.553,A -85,B 0,C 180,E1 -576.249,E2 -576.249} C_VEL
LIN {X 0,Y 601.33,Z 402.82,A -85,B 0,C 180,E1 -577.427,E2 -577.427} C_VEL
LIN {X 0,Y 601.317,Z 402.911,A -85,B 0,C 180,E1 -578.457,E2 -578.457} C_VEL
LIN {X 0,Y 601.318,Z 402.025,A -85,B 0,C 180,E1 -579.522,E2 -579.522} C_VEL
LIN {X 0,Y 601.33,Z 399.397,A -85,B 0,C 180,E1 -580.881,E2 -580.881} C_VEL
LIN {X 0,Y 601.358,Z 395.271,A -85,B 0,C 180,E1 -582.176,E2 -582.176} C_VEL
LIN {X 0,Y 601.344,Z 390.038,A -85,B 0,C 180,E1 -583.343,E2 -583.343} C_VEL
LIN {X 0,Y 601.398,Z 383.063,A -85,B 0,C 180,E1 -584.521,E2 -584.521} C_VEL
LIN {X 0,Y 601.398,Z 375.938,A -85,B 0,C 180,E1 -585.48,E2 -585.48} C_VEL
LIN {X 0,Y 601.432,Z 367.29,A -85,B 0,C 180,E1 -586.427,E2 -586.427} C_VEL
LIN {X 0,Y 601.449,Z 357.007,A -85,B 0,C 180,E1 -587.333,E2 -587.333} C_VEL
LIN {X 0,Y 601.448,Z 345.83,A -85,B 0,C 180,E1 -588.125,E2 -588.125} C_VEL
LIN {X 0,Y 601.5,Z 333.579,A -85,B 0,C 180,E1 -588.8,E2 -588.8} C_VEL
LIN {X 0,Y 601.554,Z 321.516,A -85,B 0,C 180,E1 -589.31,E2 -589.31} C_VEL
LIN {X 0,Y 601.557,Z 308.792,A -85,B 0,C 180,E1 -589.7,E2 -589.7} C_VEL
LIN {X 0,Y 601.601,Z 295.685,A -85,B 0,C 180,E1 -589.954,E2 -589.954} C_VEL
LIN {X 0,Y 601.538,Z 194.315,A -85,B 0,C 180,E1 -591.176,E2 -591.176} C_VEL
LIN {X 0,Y 601.397,Z 193.301,A -85,B 0,C 180,E1 -591.21,E2 -591.21} C_VEL
LIN {X 0,Y 601.418,Z 179.906,A -85,B 0,C 180,E1 -593.863,E2 -593.863} C_VEL
LIN {X 0,Y 601.405,Z 179.568,A -85,B 0,C 180,E1 -593.991,E2 -593.991} C_VEL
LIN {X 0,Y 601.415,Z 179.566,A -85,B 0,C 180,E1 -596.686,E2 -596.686} C_VEL
LIN {X 0,Y 601.405,Z 179.573,A -85,B 0,C 180,E1 -599.057,E2 -599.057} C_VEL
LIN {X 0,Y 601.424,Z 179.57,A -85,B 0,C 180,E1 -601.373,E2 -601.373} C_VEL
LIN {X 0,Y 601.392,Z 179.57,A -85,B 0,C 180,E1 -603.636,E2 -603.636} C_VEL
LIN {X 0,Y 601.409,Z 179.565,A -85,B 0,C 180,E1 -605.858,E2 -605.858} C_VEL
LIN {X 0,Y 601.404,Z 179.572,A -85,B 0,C 180,E1 -608.761,E2 -608.761} C_VEL
LIN {X 0,Y 601.387,Z 179.569,A -85,B 0,C 180,E1 -611.607,E2 -611.607} C_VEL
LIN {X 0,Y 601.412,Z 179.568,A -85,B 0,C 180,E1 -614.409,E2 -614.409} C_VEL
LIN {X 0,Y 601.405,Z 179.57,A -85,B 0,C 180,E1 -617.172,E2 -617.172} C_VEL
LIN {X 0,Y 601.427,Z 179.563,A -85,B 0,C 180,E1 -619.905,E2 -619.905} C_VEL
LIN {X 0,Y 601.439,Z 179.571,A -85,B 0,C 180,E1 -622.615,E2 -622.615} C_VEL
LIN {X 0,Y 601.396,Z 179.568,A -85,B 0,C 180,E1 -625.308,E2 -625.308} C_VEL
LIN {X 0,Y 601.435,Z 179.564,A -85,B 0,C 180,E1 -627.991,E2 -627.991} C_VEL
LIN {X 0,Y 601.445,Z 179.568,A -85,B 0,C 180,E1 -630.67,E2 -630.67} C_VEL
LIN {X 0,Y 601.377,Z 179.569,A -85,B 0,C 180,E1 -633.35,E2 -633.35} C_VEL
LIN {X 0,Y 601.438,Z 179.566,A -85,B 0,C 180,E1 -636.037,E2 -636.037} C_VEL
LIN {X 0,Y 601.402,Z 179.569,A -85,B 0,C 180,E1 -638.738,E2 -638.738} C_VEL
LIN {X 0,Y 601.408,Z 179.566,A -85,B 0,C 180,E1 -641.459,E2 -641.459} C_VEL
LIN {X 0,Y 601.416,Z 179.574,A -85,B 0,C 180,E1 -644.206,E2 -644.206} C_VEL
LIN {X 0,Y 601.404,Z 179.566,A -85,B 0,C 180,E1 -646.987,E2 -646.987} C_VEL
LIN {X 0,Y 601.399,Z 179.573,A -85,B 0,C 180,E1 -649.81,E2 -649.81} C_VEL
LIN {X 0,Y 601.402,Z 179.567,A -85,B 0,C 180,E1 -652.684,E2 -652.684} C_VEL
LIN {X 0,Y 601.388,Z 179.567,A -85,B 0,C 180,E1 -654.879,E2 -654.879} C_VEL
LIN {X 0,Y 601.408,Z 179.568,A -85,B 0,C 180,E1 -657.361,E2 -657.361} C_VEL
LIN {X 0,Y 601.404,Z 179.57,A -85,B 0,C 180,E1 -660.166,E2 -660.166} C_VEL
LIN {X 0,Y 601.401,Z 179.566,A -85,B 0,C 180,E1 -662.712,E2 -662.712} C_VEL
LIN {X 0,Y 601.387,Z 179.57,A -85,B 0,C 180,E1 -665.111,E2 -665.111} C_VEL
LIN {X 0,Y 601.435,Z 179.569,A -85,B 0,C 180,E1 -667.419,E2 -667.419} C_VEL
LIN {X 0,Y 601.382,Z 179.572,A -85,B 0,C 180,E1 -669.998,E2 -669.998} C_VEL
LIN {X 0,Y 601.381,Z 179.569,A -85,B 0,C 180,E1 -672.673,E2 -672.673} C_VEL
LIN {X 0,Y 601.4,Z 179.566,A -85,B 0,C 180,E1 -674.533,E2 -674.533} C_VEL
LIN {X 0,Y 601.407,Z 179.575,A -85,B 0,C 180,E1 -677.41,E2 -677.41} C_VEL
LIN {X 0,Y 601.391,Z 179.568,A -85,B 0,C 180,E1 -680.003,E2 -680.003} C_VEL
LIN {X 0,Y 601.436,Z 179.563,A -85,B 0,C 180,E1 -682.618,E2 -682.618} C_VEL
LIN {X 0,Y 601.41,Z 179.566,A -85,B 0,C 180,E1 -685.88,E2 -685.88} C_VEL
LIN {X 0,Y 601.418,Z 179.566,A -85,B 0,C 180,E1 -688.546,E2 -688.546} C_VEL
LIN {X 0,Y 601.411,Z 179.57,A -85,B 0,C 180,E1 -691.372,E2 -691.372} C_VEL
LIN {X 0,Y 601.387,Z 179.569,A -85,B 0,C 180,E1 -693.636,E2 -693.636} C_VEL
LIN {X 0,Y 601.403,Z 179.566,A -85,B 0,C 180,E1 -695.857,E2 -695.857} C_VEL
LIN {X 0,Y 601.401,Z 179.575,A -85,B 0,C 180,E1 -698.76,E2 -698.76} C_VEL
LIN {X 0,Y 601.37,Z 179.57,A -85,B 0,C 180,E1 -701.607,E2 -701.607} C_VEL
LIN {X 0,Y 601.405,Z 179.57,A -85,B 0,C 180,E1 -704.408,E2 -704.408} C_VEL
LIN {X 0,Y 601.376,Z 179.572,A -85,B 0,C 180,E1 -707.171,E2 -707.171} C_VEL
LIN {X 0,Y 601.423,Z 179.564,A -85,B 0,C 180,E1 -709.905,E2 -709.905} C_VEL
LIN {X 0,Y 601.407,Z 179.575,A -85,B 0,C 180,E1 -712.614,E2 -712.614} C_VEL
LIN {X 0,Y 601.387,Z 179.568,A -85,B 0,C 180,E1 -715.308,E2 -715.308} C_VEL
LIN {X 0,Y 601.435,Z 179.565,A -85,B 0,C 180,E1 -717.991,E2 -717.991} C_VEL
LIN {X 0,Y 601.434,Z 179.567,A -85,B 0,C 180,E1 -720.67,E2 -720.67} C_VEL
LIN {X 0,Y 601.37,Z 179.57,A -85,B 0,C 180,E1 -723.35,E2 -723.35} C_VEL
LIN {X 0,Y 601.437,Z 179.569,A -85,B 0,C 180,E1 -726.037,E2 -726.037} C_VEL
LIN {X 0,Y 601.392,Z 179.569,A -85,B 0,C 180,E1 -728.738,E2 -728.738} C_VEL
LIN {X 0,Y 601.39,Z 179.567,A -85,B 0,C 180,E1 -730.993,E2 -730.993} C_VEL
LIN {X 0,Y 601.403,Z 179.568,A -85,B 0,C 180,E1 -733.516,E2 -733.516} C_VEL
LIN {X 0,Y 601.411,Z 179.57,A -85,B 0,C 180,E1 -736.288,E2 -736.288} C_VEL
LIN {X 0,Y 601.406,Z 179.566,A -85,B 0,C 180,E1 -739.099,E2 -739.099} C_VEL
LIN {X 0,Y 601.397,Z 179.575,A -85,B 0,C 180,E1 -741.96,E2 -741.96} C_VEL
LIN {X 0,Y 601.383,Z 179.568,A -85,B 0,C 180,E1 -744.88,E2 -744.88} C_VEL
LIN {X 0,Y 601.404,Z 179.57,A -85,B 0,C 180,E1 -747.36,E2 -747.36} C_VEL
LIN {X 0,Y 601.402,Z 179.568,A -85,B 0,C 180,E1 -750.166,E2 -750.166} C_VEL
LIN {X 0,Y 601.395,Z 179.567,A -85,B 0,C 180,E1 -752.711,E2 -752.711} C_VEL
LIN {X 0,Y 601.38,Z 179.572,A -85,B 0,C 180,E1 -755.109,E2 -755.109} C_VEL
LIN {X 0,Y 601.434,Z 179.572,A -85,B 0,C 180,E1 -757.419,E2 -757.419} C_VEL
LIN {X 0,Y 601.38,Z 179.57,A -85,B 0,C 180,E1 -759.998,E2 -759.998} C_VEL
LIN {X 0,Y 601.376,Z 179.57,A -85,B 0,C 180,E1 -762.674,E2 -762.674} C_VEL
LIN {X 0,Y 601.402,Z 179.573,A -85,B 0,C 180,E1 -765.479,E2 -765.479} C_VEL
LIN {X 0,Y 601.407,Z 179.566,A -85,B 0,C 180,E1 -768.409,E2 -768.409} C_VEL
LIN {X 0,Y 601.398,Z 179.57,A -85,B 0,C 180,E1 -771.533,E2 -771.533} C_VEL
LIN {X 0,Y 601.388,Z 179.569,A -85,B 0,C 180,E1 -773.742,E2 -773.742} C_VEL
LIN {X 0,Y 601.402,Z 179.566,A -85,B 0,C 180,E1 -776.069,E2 -776.069} C_VEL
LIN {X 0,Y 601.415,Z 179.568,A -85,B 0,C 180,E1 -778.547,E2 -778.547} C_VEL
LIN {X 0,Y 601.399,Z 179.57,A -85,B 0,C 180,E1 -781.371,E2 -781.371} C_VEL
LIN {X 0,Y 601.38,Z 179.57,A -85,B 0,C 180,E1 -783.635,E2 -783.635} C_VEL
LIN {X 0,Y 601.416,Z 179.637,A -85,B 0,C 180,E1 -785.664,E2 -785.664} C_VEL
LIN {X 0,Y 601.761,Z 184.021,A -85,B 0,C 180,E1 -786.238,E2 -786.238} C_VEL
LIN {X 0,Y 601.654,Z 207.129,A -85,B 0,C 180,E1 -789.147,E2 -789.147} C_VEL
LIN {X 0,Y 601.585,Z 229.942,A -85,B 0,C 180,E1 -791.966,E2 -791.966} C_VEL
LIN {X 0,Y 601.485,Z 252.903,A -85,B 0,C 180,E1 -794.758,E2 -794.758} C_VEL
LIN {X 0,Y 601.478,Z 270.229,A -85,B 0,C 180,E1 -796.819,E2 -796.819} C_VEL
LIN {X 0,Y 601.62,Z 378.935,A -85,B 0,C 180,E1 -798.139,E2 -798.139} C_VEL
LIN {X 0,Y 601.56,Z 392.21,A -85,B 0,C 180,E1 -798.437,E2 -798.437} C_VEL
LIN {X 0,Y 601.546,Z 403.9,A -85,B 0,C 180,E1 -798.825,E2 -798.825} C_VEL
LIN {X 0,Y 601.522,Z 416.629,A -85,B 0,C 180,E1 -799.396,E2 -799.396} C_VEL
LIN {X 0,Y 601.483,Z 428.196,A -85,B 0,C 180,E1 -800.076,E2 -800.076} C_VEL
LIN {X 0,Y 601.444,Z 438.593,A -85,B 0,C 180,E1 -800.839,E2 -800.839} C_VEL
LIN {X 0,Y 601.429,Z 447.11,A -85,B 0,C 180,E1 -801.601,E2 -801.601} C_VEL
LIN {X 0,Y 601.418,Z 454.959,A -85,B 0,C 180,E1 -802.446,E2 -802.446} C_VEL
LIN {X 0,Y 601.37,Z 462.224,A -85,B 0,C 180,E1 -803.398,E2 -803.398} C_VEL
LIN {X 0,Y 601.372,Z 467.865,A -85,B 0,C 180,E1 -804.299,E2 -804.299} C_VEL
LIN {X 0,Y 601.336,Z 472.949,A -85,B 0,C 180,E1 -805.307,E2 -805.307} C_VEL
LIN {X 0,Y 601.368,Z 476.895,A -85,B 0,C 180,E1 -806.314,E2 -806.314} C_VEL
LIN {X 0,Y 601.325,Z 479.808,A -85,B 0,C 180,E1 -807.32,E2 -807.32} C_VEL
LIN {X 0,Y 601.343,Z 481.201,A -85,B 0,C 180,E1 -807.991,E2 -807.991} C_VEL
LIN {X 0,Y 601.339,Z 482.784,A -85,B 0,C 180,E1 -809.33,E2 -809.33} C_VEL
LIN {X 0,Y 601.335,Z 483,A -85,B 0,C 180,E1 -810,E2 -810} C_VEL
LIN {X 0,Y 601.347,Z 482.185,A -85,B 0,C 180,E1 -811.339,E2 -811.339} C_VEL
LIN {X 0,Y 601.343,Z 481.202,A -85,B 0,C 180,E1 -812.009,E2 -812.009} C_VEL
LIN {X 0,Y 601.325,Z 479.81,A -85,B 0,C 180,E1 -812.679,E2 -812.679} C_VEL
LIN {X 0,Y 601.368,Z 476.897,A -85,B 0,C 180,E1 -813.685,E2 -813.685} C_VEL
LIN {X 0,Y 601.336,Z 472.95,A -85,B 0,C 180,E1 -814.693,E2 -814.693} C_VEL
LIN {X 0,Y 601.373,Z 466.878,A -85,B 0,C 180,E1 -815.869,E2 -815.869} C_VEL
LIN {X 0,Y 601.382,Z 460.237,A -85,B 0,C 180,E1 -816.88,E2 -816.88} C_VEL
LIN {X 0,Y 601.4,Z 451.991,A -85,B 0,C 180,E1 -817.892,E2 -817.892} C_VEL
LIN {X 0,Y 601.436,Z 443.539,A -85,B 0,C 180,E1 -818.737,E2 -818.737} C_VEL
LIN {X 0,Y 601.449,Z 433.095,A -85,B 0,C 180,E1 -819.585,E2 -819.585} C_VEL
LIN {X 0,Y 601.467,Z 422.76,A -85,B 0,C 180,E1 -820.264,E2 -820.264} C_VEL
LIN {X 0,Y 601.537,Z 410.598,A -85,B 0,C 180,E1 -820.896,E2 -820.896} C_VEL
LIN {X 0,Y 601.555,Z 398.222,A -85,B 0,C 180,E1 -821.379,E2 -821.379} C_VEL
LIN {X 0,Y 601.582,Z 385.444,A -85,B 0,C 180,E1 -821.733,E2 -821.733} C_VEL
LIN {X 0,Y 601.62,Z 373.096,A -85,B 0,C 180,E1 -821.946,E2 -821.946} C_VEL
LIN {X 0,Y 601.477,Z 270.261,A -85,B 0,C 180,E1 -823.181,E2 -823.181} C_VEL
LIN {X 0,Y 601.543,Z 248.601,A -85,B 0,C 180,E1 -825.762,E2 -825.762} C_VEL
LIN {X 0,Y 601.603,Z 224.062,A -85,B 0,C 180,E1 -828.757,E2 -828.757} C_VEL
LIN {X 0,Y 601.698,Z 201.245,A -85,B 0,C 180,E1 -831.588,E2 -831.588} C_VEL
LIN {X 0,Y 601.717,Z 181.154,A -85,B 0,C 180,E1 -834.129,E2 -834.129} C_VEL
LIN {X 0,Y 601.387,Z 179.573,A -85,B 0,C 180,E1 -834.376,E2 -834.376} C_VEL
LIN {X 0,Y 601.452,Z 179.57,A -85,B 0,C 180,E1 -837.111,E2 -837.111} C_VEL
LIN {X 0,Y 601.386,Z 179.573,A -85,B 0,C 180,E1 -839.395,E2 -839.395} C_VEL
LIN {X 0,Y 601.385,Z 179.569,A -85,B 0,C 180,E1 -841.728,E2 -841.728} C_VEL
LIN {X 0,Y 601.405,Z 179.566,A -85,B 0,C 180,E1 -844.12,E2 -844.12} C_VEL
LIN {X 0,Y 601.435,Z 179.564,A -85,B 0,C 180,E1 -847.382,E2 -847.382} C_VEL
LIN {X 0,Y 601.378,Z 179.57,A -85,B 0,C 180,E1 -849.998,E2 -849.998} C_VEL
LIN {X 0,Y 601.406,Z 179.576,A -85,B 0,C 180,E1 -852.671,E2 -852.671} C_VEL
LIN {X 0,Y 601.399,Z 179.566,A -85,B 0,C 180,E1 -855.479,E2 -855.479} C_VEL
LIN {X 0,Y 601.419,Z 179.572,A -85,B 0,C 180,E1 -858.407,E2 -858.407} C_VEL
LIN {X 0,Y 601.406,Z 179.569,A -85,B 0,C 180,E1 -860.873,E2 -860.873} C_VEL
LIN {X 0,Y 601.392,Z 179.567,A -85,B 0,C 180,E1 -863.416,E2 -863.416} C_VEL
LIN {X 0,Y 601.428,Z 179.569,A -85,B 0,C 180,E1 -866.065,E2 -866.065} C_VEL
LIN {X 0,Y 601.398,Z 179.567,A -85,B 0,C 180,E1 -869.057,E2 -869.057} C_VEL
LIN {X 0,Y 601.403,Z 179.566,A -85,B 0,C 180,E1 -871.372,E2 -871.372} C_VEL
LIN {X 0,Y 601.411,Z 179.574,A -85,B 0,C 180,E1 -874.133,E2 -874.133} C_VEL
LIN {X 0,Y 601.392,Z 179.569,A -85,B 0,C 180,E1 -876.588,E2 -876.588} C_VEL
LIN {X 0,Y 601.415,Z 179.568,A -85,B 0,C 180,E1 -879.477,E2 -879.477} C_VEL
LIN {X 0,Y 601.389,Z 179.571,A -85,B 0,C 180,E1 -882.311,E2 -882.311} C_VEL
LIN {X 0,Y 601.404,Z 179.567,A -85,B 0,C 180,E1 -884.408,E2 -884.408} C_VEL
LIN {X 0,Y 601.406,Z 179.568,A -85,B 0,C 180,E1 -887.171,E2 -887.171} C_VEL
LIN {X 0,Y 601.437,Z 179.567,A -85,B 0,C 180,E1 -889.905,E2 -889.905} C_VEL
LIN {X 0,Y 601.401,Z 179.566,A -85,B 0,C 180,E1 -892.614,E2 -892.614} C_VEL
LIN {X 0,Y 601.424,Z 179.571,A -85,B 0,C 180,E1 -895.308,E2 -895.308} C_VEL
LIN {X 0,Y 601.439,Z 179.563,A -85,B 0,C 180,E1 -897.991,E2 -897.991} C_VEL
LIN {X 0,Y 601.431,Z 179.564,A -85,B 0,C 180,E1 -900.669,E2 -900.669} C_VEL
LIN {X 0,Y 601.432,Z 179.571,A -85,B 0,C 180,E1 -903.349,E2 -903.349} C_VEL
LIN {X 0,Y 601.435,Z 179.562,A -85,B 0,C 180,E1 -906.037,E2 -906.037} C_VEL
LIN {X 0,Y 601.404,Z 179.57,A -85,B 0,C 180,E1 -908.738,E2 -908.738} C_VEL
LIN {X 0,Y 601.437,Z 179.566,A -85,B 0,C 180,E1 -911.458,E2 -911.458} C_VEL
LIN {X 0,Y 601.403,Z 179.568,A -85,B 0,C 180,E1 -912.354,E2 -912.354} C_VEL
LIN {X 0,Y 600.735,Z 179.659,A -85,B 0,C 180,E1 -912.914,E2 -912.914} C_VEL
LIN {X 0,Y 597.888,Z 180.016,A -85,B 0,C 180,E1 -913.822,E2 -913.822} C_VEL
LIN {X 0,Y 595.481,Z 180.315,A -85,B 0,C 180,E1 -914.552,E2 -914.552} C_VEL
LIN {X 0,Y 594.444,Z 180.441,A -85,B 0,C 180,E1 -915.115,E2 -915.115} C_VEL
LIN {X 0,Y 594.357,Z 180.448,A -85,B 0,C 180,E1 -915.306,E2 -915.306} C_VEL
LIN {X 0,Y 594.382,Z 180.446,A -85,B 0,C 180,E1 -917.194,E2 -917.194} C_VEL
LIN {X 0,Y 594.369,Z 180.443,A -85,B 0,C 180,E1 -920.054,E2 -920.054} C_VEL
LIN {X 0,Y 594.386,Z 180.547,A -85,B 0,C 180,E1 -922.164,E2 -922.164} C_VEL
LIN {X 0,Y 594.368,Z 193.375,A -85,B 0,C 180,E1 -924.736,E2 -924.736} C_VEL
LIN {X 0,Y 594.76,Z 198.293,A -85,B 0,C 180,E1 -924.81,E2 -924.81} C_VEL
LIN {X 0,Y 594.657,Z 299.516,A -85,B 0,C 180,E1 -926.055,E2 -926.055} C_VEL
LIN {X 0,Y 594.607,Z 312.712,A -85,B 0,C 180,E1 -926.36,E2 -926.36} C_VEL
LIN {X 0,Y 594.576,Z 325.138,A -85,B 0,C 180,E1 -926.785,E2 -926.785} C_VEL
LIN {X 0,Y 594.494,Z 337.464,A -85,B 0,C 180,E1 -927.36,E2 -927.36} C_VEL
LIN {X 0,Y 594.428,Z 348.703,A -85,B 0,C 180,E1 -928.036,E2 -928.036} C_VEL
LIN {X 0,Y 594.421,Z 358.742,A -85,B 0,C 180,E1 -928.786,E2 -928.786} C_VEL
LIN {X 0,Y 594.377,Z 367.482,A -85,B 0,C 180,E1 -929.581,E2 -929.581} C_VEL
LIN {X 0,Y 594.322,Z 376.27,A -85,B 0,C 180,E1 -930.563,E2 -930.563} C_VEL
LIN {X 0,Y 594.326,Z 384.001,A -85,B 0,C 180,E1 -931.635,E2 -931.635} C_VEL
LIN {X 0,Y 594.269,Z 389.186,A -85,B 0,C 180,E1 -932.523,E2 -932.523} C_VEL
LIN {X 0,Y 594.268,Z 394.915,A -85,B 0,C 180,E1 -933.768,E2 -933.768} C_VEL
LIN {X 0,Y 594.255,Z 397.75,A -85,B 0,C 180,E1 -934.588,E2 -934.588} C_VEL
LIN {X 0,Y 594.227,Z 400,A -85,B 0,C 180,E1 -935.417,E2 -935.417} C_VEL
LIN {X 0,Y 594.221,Z 401.919,A -85,B 0,C 180,E1 -936.462,E2 -936.462} C_VEL
LIN {X 0,Y 594.227,Z 402.901,A -85,B 0,C 180,E1 -937.588,E2 -937.588} C_VEL
LIN {X 0,Y 594.208,Z 402.718,A -85,B 0,C 180,E1 -938.819,E2 -938.819} C_VEL
LIN {X 0,Y 594.23,Z 401.722,A -85,B 0,C 180,E1 -939.758,E2 -939.758} C_VEL
LIN {X 0,Y 594.23,Z 399.683,A -85,B 0,C 180,E1 -940.806,E2 -940.806} C_VEL
LIN {X 0,Y 594.262,Z 395.779,A -85,B 0,C 180,E1 -942.086,E2 -942.086} C_VEL
LIN {X 0,Y 594.275,Z 390.538,A -85,B 0,C 180,E1 -943.308,E2 -943.308} C_VEL
LIN {X 0,Y 594.308,Z 385.341,A -85,B 0,C 180,E1 -944.243,E2 -944.243} C_VEL
LIN {X 0,Y 594.32,Z 377.79,A -85,B 0,C 180,E1 -945.336,E2 -945.336} C_VEL
LIN {X 0,Y 594.345,Z 369.512,A -85,B 0,C 180,E1 -946.298,E2 -946.298} C_VEL
LIN {X 0,Y 594.385,Z 359.643,A -85,B 0,C 180,E1 -947.23,E2 -947.23} C_VEL
LIN {X 0,Y 594.453,Z 348.542,A -85,B 0,C 180,E1 -948.065,E2 -948.065} C_VEL
LIN {X 0,Y 594.505,Z 337.722,A -85,B 0,C 180,E1 -948.716,E2 -948.716} C_VEL
LIN {X 0,Y 594.57,Z 326.022,A -85,B 0,C 180,E1 -949.27,E2 -949.27} C_VEL
LIN {X 0,Y 594.608,Z 313.128,A -85,B 0,C 180,E1 -949.719,E2 -949.719} C_VEL
LIN {X 0,Y 594.651,Z 300.108,A -85,B 0,C 180,E1 -950.024,E2 -950.024} C_VEL
LIN {X 0,Y 594.698,Z 252.813,A -85,B 0,C 180,E1 -950.62,E2 -950.62} C_VEL
LIN {X 0,Y 594.664,Z 195.305,A -85,B 0,C 180,E1 -951.319,E2 -951.319} C_VEL
LIN {X 0,Y 594.335,Z 193.378,A -85,B 0,C 180,E1 -951.354,E2 -951.354} C_VEL
LIN {X 0,Y 594.377,Z 180.474,A -85,B 0,C 180,E1 -953.941,E2 -953.941} C_VEL
LIN {X 0,Y 594.364,Z 180.443,A -85,B 0,C 180,E1 -956.238,E2 -956.238} C_VEL
LIN {X 0,Y 594.367,Z 180.444,A -85,B 0,C 180,E1 -958.65,E2 -958.65} C_VEL
LIN {X 0,Y 594.382,Z 180.448,A -85,B 0,C 180,E1 -961.043,E2 -961.043} C_VEL
LIN {X 0,Y 594.381,Z 180.448,A -85,B 0,C 180,E1 -963.3,E2 -963.3} C_VEL
LIN {X 0,Y 594.347,Z 180.447,A -85,B 0,C 180,E1 -965.575,E2 -965.575} C_VEL
LIN {X 0,Y 594.359,Z 180.446,A -85,B 0,C 180,E1 -968.497,E2 -968.497} C_VEL
LIN {X 0,Y 594.366,Z 180.446,A -85,B 0,C 180,E1 -971.382,E2 -971.382} C_VEL
LIN {X 0,Y 594.36,Z 180.444,A -85,B 0,C 180,E1 -974.219,E2 -974.219} C_VEL
LIN {X 0,Y 594.356,Z 180.45,A -85,B 0,C 180,E1 -977.017,E2 -977.017} C_VEL
LIN {X 0,Y 594.384,Z 180.44,A -85,B 0,C 180,E1 -979.784,E2 -979.784} C_VEL
LIN {X 0,Y 594.393,Z 180.447,A -85,B 0,C 180,E1 -982.527,E2 -982.527} C_VEL
LIN {X 0,Y 594.369,Z 180.443,A -85,B 0,C 180,E1 -985.252,E2 -985.252} C_VEL
LIN {X 0,Y 594.404,Z 180.439,A -85,B 0,C 180,E1 -987.967,E2 -987.967} C_VEL
LIN {X 0,Y 594.416,Z 180.443,A -85,B 0,C 180,E1 -990.678,E2 -990.678} C_VEL
LIN {X 0,Y 594.332,Z 180.447,A -85,B 0,C 180,E1 -993.39,E2 -993.39} C_VEL
LIN {X 0,Y 594.385,Z 180.446,A -85,B 0,C 180,E1 -996.109,E2 -996.109} C_VEL
LIN {X 0,Y 594.369,Z 180.444,A -85,B 0,C 180,E1 -998.843,E2 -998.843} C_VEL
LIN {X 0,Y 594.378,Z 180.442,A -85,B 0,C 180,E1 -1001.596,E2 -1001.596} C_VEL
LIN {X 0,Y 594.383,Z 180.447,A -85,B 0,C 180,E1 -1004.377,E2 -1004.377} C_VEL
LIN {X 0,Y 594.372,Z 180.442,A -85,B 0,C 180,E1 -1007.194,E2 -1007.194} C_VEL
LIN {X 0,Y 594.365,Z 180.453,A -85,B 0,C 180,E1 -1010.054,E2 -1010.054} C_VEL
LIN {X 0,Y 594.352,Z 180.444,A -85,B 0,C 180,E1 -1012.968,E2 -1012.968} C_VEL
LIN {X 0,Y 594.37,Z 180.443,A -85,B 0,C 180,E1 -1015.194,E2 -1015.194} C_VEL
LIN {X 0,Y 594.352,Z 180.449,A -85,B 0,C 180,E1 -1017.52,E2 -1017.52} C_VEL
LIN {X 0,Y 594.369,Z 180.444,A -85,B 0,C 180,E1 -1020.325,E2 -1020.325} C_VEL
LIN {X 0,Y 594.376,Z 180.442,A -85,B 0,C 180,E1 -1022.951,E2 -1022.951} C_VEL
LIN {X 0,Y 594.348,Z 180.451,A -85,B 0,C 180,E1 -1025.409,E2 -1025.409} C_VEL
LIN {X 0,Y 594.373,Z 180.446,A -85,B 0,C 180,E1 -1027.942,E2 -1027.942} C_VEL
LIN {X 0,Y 594.375,Z 180.442,A -85,B 0,C 180,E1 -1030.822,E2 -1030.822} C_VEL
LIN {X 0,Y 594.362,Z 180.447,A -85,B 0,C 180,E1 -1033.839,E2 -1033.839} C_VEL
LIN {X 0,Y 594.352,Z 180.445,A -85,B 0,C 180,E1 -1036.699,E2 -1036.699} C_VEL
LIN {X 0,Y 594.36,Z 180.452,A -85,B 0,C 180,E1 -1039.432,E2 -1039.432} C_VEL
LIN {X 0,Y 594.385,Z 180.44,A -85,B 0,C 180,E1 -1042.393,E2 -1042.393} C_VEL
LIN {X 0,Y 594.378,Z 180.447,A -85,B 0,C 180,E1 -1045.42,E2 -1045.42} C_VEL
LIN {X 0,Y 594.371,Z 180.442,A -85,B 0,C 180,E1 -1048.359,E2 -1048.359} C_VEL
LIN {X 0,Y 594.377,Z 180.452,A -85,B 0,C 180,E1 -1051.044,E2 -1051.044} C_VEL
LIN {X 0,Y 594.38,Z 180.446,A -85,B 0,C 180,E1 -1053.3,E2 -1053.3} C_VEL
LIN {X 0,Y 594.342,Z 180.447,A -85,B 0,C 180,E1 -1055.577,E2 -1055.577} C_VEL
LIN {X 0,Y 594.357,Z 180.448,A -85,B 0,C 180,E1 -1058.496,E2 -1058.496} C_VEL
LIN {X 0,Y 594.352,Z 180.446,A -85,B 0,C 180,E1 -1061.382,E2 -1061.382} C_VEL
LIN {X 0,Y 594.37,Z 180.442,A -85,B 0,C 180,E1 -1063.514,E2 -1063.514} C_VEL
LIN {X 0,Y 594.37,Z 180.446,A -85,B 0,C 180,E1 -1066.321,E2 -1066.321} C_VEL
LIN {X 0,Y 594.351,Z 180.447,A -85,B 0,C 180,E1 -1069.094,E2 -1069.094} C_VEL
LIN {X 0,Y 594.376,Z 180.442,A -85,B 0,C 180,E1 -1071.843,E2 -1071.843} C_VEL
LIN {X 0,Y 594.383,Z 180.449,A -85,B 0,C 180,E1 -1074.572,E2 -1074.572} C_VEL
LIN {X 0,Y 594.378,Z 180.441,A -85,B 0,C 180,E1 -1077.289,E2 -1077.289} C_VEL
LIN {X 0,Y 594.415,Z 180.441,A -85,B 0,C 180,E1 -1080,E2 -1080} C_VEL
LIN {X 0,Y 594.387,Z 180.443,A -85,B 0,C 180,E1 -1082.711,E2 -1082.711} C_VEL
LIN {X 0,Y 594.371,Z 180.442,A -85,B 0,C 180,E1 -1085.428,E2 -1085.428} C_VEL
LIN {X 0,Y 594.381,Z 180.451,A -85,B 0,C 180,E1 -1088.157,E2 -1088.157} C_VEL
LIN {X 0,Y 594.368,Z 180.442,A -85,B 0,C 180,E1 -1091.061,E2 -1091.061} C_VEL
LIN {X 0,Y 594.372,Z 180.446,A -85,B 0,C 180,E1 -1093.679,E2 -1093.679} C_VEL
LIN {X 0,Y 594.335,Z 180.447,A -85,B 0,C 180,E1 -1096.699,E2 -1096.699} C_VEL
LIN {X 0,Y 594.359,Z 180.445,A -85,B 0,C 180,E1 -1099.335,E2 -1099.335} C_VEL
LIN {X 0,Y 594.355,Z 180.448,A -85,B 0,C 180,E1 -1101.504,E2 -1101.504} C_VEL
LIN {X 0,Y 594.346,Z 180.446,A -85,B 0,C 180,E1 -1104.448,E2 -1104.448} C_VEL
LIN {X 0,Y 594.36,Z 180.443,A -85,B 0,C 180,E1 -1106.701,E2 -1106.701} C_VEL
LIN {X 0,Y 594.357,Z 180.452,A -85,B 0,C 180,E1 -1109.778,E2 -1109.778} C_VEL
LIN {X 0,Y 594.344,Z 180.447,A -85,B 0,C 180,E1 -1112.149,E2 -1112.149} C_VEL
LIN {X 0,Y 594.362,Z 180.443,A -85,B 0,C 180,E1 -1114.581,E2 -1114.581} C_VEL
LIN {X 0,Y 594.385,Z 180.448,A -85,B 0,C 180,E1 -1117.607,E2 -1117.607} C_VEL
LIN {X 0,Y 594.362,Z 180.443,A -85,B 0,C 180,E1 -1120.568,E2 -1120.568} C_VEL
LIN {X 0,Y 594.346,Z 180.455,A -85,B 0,C 180,E1 -1123.302,E2 -1123.302} C_VEL
LIN {X 0,Y 594.344,Z 180.445,A -85,B 0,C 180,E1 -1126.163,E2 -1126.163} C_VEL
LIN {X 0,Y 594.371,Z 180.452,A -85,B 0,C 180,E1 -1129.179,E2 -1129.179} C_VEL
LIN {X 0,Y 594.367,Z 180.442,A -85,B 0,C 180,E1 -1132.058,E2 -1132.058} C_VEL
LIN {X 0,Y 594.328,Z 180.451,A -85,B 0,C 180,E1 -1134.68,E2 -1134.68} C_VEL
LIN {X 0,Y 594.374,Z 180.451,A -85,B 0,C 180,E1 -1137.09,E2 -1137.09} C_VEL
LIN {X 0,Y 594.35,Z 180.445,A -85,B 0,C 180,E1 -1139.678,E2 -1139.678} C_VEL
LIN {X 0,Y 594.322,Z 180.449,A -85,B 0,C 180,E1 -1141.77,E2 -1141.77} C_VEL
LIN {X 0,Y 594.341,Z 180.447,A -85,B 0,C 180,E1 -1144.054,E2 -1144.054} C_VEL
LIN {X 0,Y 594.368,Z 180.506,A -85,B 0,C 180,E1 -1145.469,E2 -1145.469} C_VEL
LIN {X 0,Y 594.911,Z 184.021,A -85,B 0,C 180,E1 -1145.948,E2 -1145.948} C_VEL
LIN {X 0,Y 594.754,Z 206.498,A -85,B 0,C 180,E1 -1148.813,E2 -1148.813} C_VEL
LIN {X 0,Y 594.642,Z 227.072,A -85,B 0,C 180,E1 -1151.391,E2 -1151.391} C_VEL
LIN {X 0,Y 594.566,Z 250.033,A -85,B 0,C 180,E1 -1154.224,E2 -1154.224} C_VEL
LIN {X 0,Y 594.46,Z 270.229,A -85,B 0,C 180,E1 -1156.66,E2 -1156.66} C_VEL
LIN {X 0,Y 594.745,Z 276.49,A -85,B 0,C 180,E1 -1156.743,E2 -1156.743} C_VEL
LIN {X 0,Y 594.691,Z 378.935,A -85,B 0,C 180,E1 -1157.999,E2 -1157.999} C_VEL
LIN {X 0,Y 594.602,Z 392.211,A -85,B 0,C 180,E1 -1158.3,E2 -1158.3} C_VEL
LIN {X 0,Y 594.591,Z 405.273,A -85,B 0,C 180,E1 -1158.745,E2 -1158.745} C_VEL
LIN {X 0,Y 594.536,Z 416.628,A -85,B 0,C 180,E1 -1159.27,E2 -1159.27} C_VEL
LIN {X 0,Y 594.477,Z 428.198,A -85,B 0,C 180,E1 -1159.957,E2 -1159.957} C_VEL
LIN {X 0,Y 594.414,Z 438.594,A -85,B 0,C 180,E1 -1160.729,E2 -1160.729} C_VEL
LIN {X 0,Y 594.383,Z 447.11,A -85,B 0,C 180,E1 -1161.5,E2 -1161.5} C_VEL
LIN {X 0,Y 594.347,Z 454.959,A -85,B 0,C 180,E1 -1162.355,E2 -1162.355} C_VEL
LIN {X 0,Y 594.283,Z 462.812,A -85,B 0,C 180,E1 -1163.408,E2 -1163.408} C_VEL
LIN {X 0,Y 594.289,Z 469.679,A -85,B 0,C 180,E1 -1164.571,E2 -1164.571} C_VEL
LIN {X 0,Y 594.27,Z 474.371,A -85,B 0,C 180,E1 -1165.591,E2 -1165.591} C_VEL
LIN {X 0,Y 594.267,Z 477.956,A -85,B 0,C 180,E1 -1166.61,E2 -1166.61} C_VEL
LIN {X 0,Y 594.225,Z 479.808,A -85,B 0,C 180,E1 -1167.288,E2 -1167.288} C_VEL
LIN {X 0,Y 594.242,Z 481.201,A -85,B 0,C 180,E1 -1167.967,E2 -1167.967} C_VEL
LIN {X 0,Y 594.239,Z 482.784,A -85,B 0,C 180,E1 -1169.322,E2 -1169.322} C_VEL
LIN {X 0,Y 594.236,Z 483,A -85,B 0,C 180,E1 -1170,E2 -1170} C_VEL
LIN {X 0,Y 594.247,Z 482.185,A -85,B 0,C 180,E1 -1171.355,E2 -1171.355} C_VEL
LIN {X 0,Y 594.242,Z 481.202,A -85,B 0,C 180,E1 -1172.033,E2 -1172.033} C_VEL
LIN {X 0,Y 594.226,Z 479.81,A -85,B 0,C 180,E1 -1172.711,E2 -1172.711} C_VEL
LIN {X 0,Y 594.289,Z 476.897,A -85,B 0,C 180,E1 -1173.729,E2 -1173.729} C_VEL
LIN {X 0,Y 594.241,Z 472.95,A -85,B 0,C 180,E1 -1174.749,E2 -1174.749} C_VEL
LIN {X 0,Y 594.305,Z 466.879,A -85,B 0,C 180,E1 -1175.939,E2 -1175.939} C_VEL
LIN {X 0,Y 594.308,Z 460.238,A -85,B 0,C 180,E1 -1176.962,E2 -1176.962} C_VEL
LIN {X 0,Y 594.359,Z 451.991,A -85,B 0,C 180,E1 -1177.986,E2 -1177.986} C_VEL
LIN {X 0,Y 594.382,Z 443.539,A -85,B 0,C 180,E1 -1178.842,E2 -1178.842} C_VEL
LIN {X 0,Y 594.432,Z 433.097,A -85,B 0,C 180,E1 -1179.699,E2 -1179.699} C_VEL
LIN {X 0,Y 594.481,Z 422.761,A -85,B 0,C 180,E1 -1180.386,E2 -1180.386} C_VEL
LIN {X 0,Y 594.558,Z 411.725,A -85,B 0,C 180,E1 -1180.973,E2 -1180.973} C_VEL
LIN {X 0,Y 594.579,Z 399.715,A -85,B 0,C 180,E1 -1181.464,E2 -1181.464} C_VEL
LIN {X 0,Y 594.632,Z 386.357,A -85,B 0,C 180,E1 -1181.85,E2 -1181.85} C_VEL
LIN {X 0,Y 594.69,Z 373.096,A -85,B 0,C 180,E1 -1182.087,E2 -1182.087} C_VEL
LIN {X 0,Y 594.578,Z 271.155,A -85,B 0,C 180,E1 -1183.326,E2 -1183.326} C_VEL
LIN {X 0,Y 594.445,Z 269.768,A -85,B 0,C 180,E1 -1183.372,E2 -1183.372} C_VEL
LIN {X 0,Y 594.539,Z 245.731,A -85,B 0,C 180,E1 -1186.305,E2 -1186.305} C_VEL
LIN {X 0,Y 594.676,Z 223.066,A -85,B 0,C 180,E1 -1189.108,E2 -1189.108} C_VEL
LIN {X 0,Y 594.804,Z 201.245,A -85,B 0,C 180,E1 -1191.851,E2 -1191.851} C_VEL
LIN {X 0,Y 594.89,Z 182.961,A -85,B 0,C 180,E1 -1194.19,E2 -1194.19} C_VEL
LIN {X 0,Y 594.354,Z 180.45,A -85,B 0,C 180,E1 -1194.573,E2 -1194.573} C_VEL
LIN {X 0,Y 594.377,Z 180.446,A -85,B 0,C 180,E1 -1197.461,E2 -1197.461} C_VEL
LIN {X 0,Y 594.349,Z 180.446,A -85,B 0,C 180,E1 -1200.321,E2 -1200.321} C_VEL
LIN {X 0,Y 594.373,Z 180.452,A -85,B 0,C 180,E1 -1202.95,E2 -1202.95} C_VEL
LIN {X 0,Y 594.346,Z 180.447,A -85,B 0,C 180,E1 -1205.409,E2 -1205.409} C_VEL
LIN {X 0,Y 594.368,Z 180.442,A -85,B 0,C 180,E1 -1207.942,E2 -1207.942} C_VEL
LIN {X 0,Y 594.37,Z 180.451,A -85,B 0,C 180,E1 -1210.821,E2 -1210.821} C_VEL
LIN {X 0,Y 594.35,Z 180.446,A -85,B 0,C 180,E1 -1213.301,E2 -1213.301} C_VEL
LIN {X 0,Y 594.36,Z 180.447,A -85,B 0,C 180,E1 -1216.161,E2 -1216.161} C_VEL
LIN {X 0,Y 594.374,Z 180.442,A -85,B 0,C 180,E1 -1219.178,E2 -1219.178} C_VEL
LIN {X 0,Y 594.372,Z 180.446,A -85,B 0,C 180,E1 -1222.058,E2 -1222.058} C_VEL
LIN {X 0,Y 594.349,Z 180.449,A -85,B 0,C 180,E1 -1224.677,E2 -1224.677} C_VEL
LIN {X 0,Y 594.373,Z 180.442,A -85,B 0,C 180,E1 -1227.089,E2 -1227.089} C_VEL
LIN {X 0,Y 594.367,Z 180.445,A -85,B 0,C 180,E1 -1229.675,E2 -1229.675} C_VEL
LIN {X 0,Y 594.376,Z 180.445,A -85,B 0,C 180,E1 -1232.539,E2 -1232.539} C_VEL
LIN {X 0,Y 594.371,Z 180.443,A -85,B 0,C 180,E1 -1234.807,E2 -1234.807} C_VEL
LIN {X 0,Y 594.357,Z 180.444,A -85,B 0,C 180,E1 -1237.267,E2 -1237.267} C_VEL
LIN {X 0,Y 594.367,Z 180.452,A -85,B 0,C 180,E1 -1239.946,E2 -1239.946} C_VEL
LIN {X 0,Y 594.373,Z 180.441,A -85,B 0,C 180,E1 -1242.806,E2 -1242.806} C_VEL
LIN {X 0,Y 594.388,Z 180.449,A -85,B 0,C 180,E1 -1245.827,E2 -1245.827} C_VEL
LIN {X 0,Y 594.378,Z 180.442,A -85,B 0,C 180,E1 -1248.404,E2 -1248.404} C_VEL
LIN {X 0,Y 594.374,Z 180.445,A -85,B 0,C 180,E1 -1251.158,E2 -1251.158} C_VEL
LIN {X 0,Y 594.394,Z 180.443,A -85,B 0,C 180,E1 -1253.891,E2 -1253.891} C_VEL
LIN {X 0,Y 594.361,Z 180.443,A -85,B 0,C 180,E1 -1256.611,E2 -1256.611} C_VEL
LIN {X 0,Y 594.422,Z 180.445,A -85,B 0,C 180,E1 -1259.323,E2 -1259.323} C_VEL
LIN {X 0,Y 594.405,Z 180.439,A -85,B 0,C 180,E1 -1262.033,E2 -1262.033} C_VEL
LIN {X 0,Y 594.378,Z 180.444,A -85,B 0,C 180,E1 -1264.748,E2 -1264.748} C_VEL
LIN {X 0,Y 594.395,Z 180.444,A -85,B 0,C 180,E1 -1267.473,E2 -1267.473} C_VEL
LIN {X 0,Y 594.389,Z 180.44,A -85,B 0,C 180,E1 -1270.216,E2 -1270.216} C_VEL
LIN {X 0,Y 594.36,Z 180.454,A -85,B 0,C 180,E1 -1272.983,E2 -1272.983} C_VEL
LIN {X 0,Y 594.357,Z 180.448,A -85,B 0,C 180,E1 -1275.306,E2 -1275.306} C_VEL
LIN {X 0,Y 593.68,Z 180.531,A -85,B 0,C 180,E1 -1275.872,E2 -1275.872} C_VEL
LIN {X 0,Y 590.81,Z 180.895,A -85,B 0,C 180,E1 -1276.79,E2 -1276.79} C_VEL
LIN {X 0,Y 588.399,Z 181.19,A -85,B 0,C 180,E1 -1277.529,E2 -1277.529} C_VEL
LIN {X 0,Y 587.377,Z 181.315,A -85,B 0,C 180,E1 -1278.099,E2 -1278.099} C_VEL
LIN {X 0,Y 587.301,Z 181.325,A -85,B 0,C 180,E1 -1278.292,E2 -1278.292} C_VEL
LIN {X 0,Y 587.331,Z 181.326,A -85,B 0,C 180,E1 -1281.038,E2 -1281.038} C_VEL
LIN {X 0,Y 587.329,Z 181.407,A -85,B 0,C 180,E1 -1282.144,E2 -1282.144} C_VEL
LIN {X 0,Y 587.321,Z 193.375,A -85,B 0,C 180,E1 -1284.573,E2 -1284.573} C_VEL
LIN {X 0,Y 587.866,Z 199.083,A -85,B 0,C 180,E1 -1284.662,E2 -1284.662} C_VEL
LIN {X 0,Y 587.719,Z 299.092,A -85,B 0,C 180,E1 -1285.903,E2 -1285.903} C_VEL
LIN {X 0,Y 587.652,Z 312.3,A -85,B 0,C 180,E1 -1286.207,E2 -1286.207} C_VEL
LIN {X 0,Y 587.612,Z 325.095,A -85,B 0,C 180,E1 -1286.648,E2 -1286.648} C_VEL
LIN {X 0,Y 587.501,Z 337.451,A -85,B 0,C 180,E1 -1287.23,E2 -1287.23} C_VEL
LIN {X 0,Y 587.414,Z 348.654,A -85,B 0,C 180,E1 -1287.911,E2 -1287.911} C_VEL
LIN {X 0,Y 587.406,Z 358.78,A -85,B 0,C 180,E1 -1288.678,E2 -1288.678} C_VEL
LIN {X 0,Y 587.328,Z 368.426,A -85,B 0,C 180,E1 -1289.578,E2 -1289.578} C_VEL
LIN {X 0,Y 587.272,Z 376.479,A -85,B 0,C 180,E1 -1290.499,E2 -1290.499} C_VEL
LIN {X 0,Y 587.242,Z 384.107,A -85,B 0,C 180,E1 -1291.574,E2 -1291.574} C_VEL
LIN {X 0,Y 587.175,Z 389.885,A -85,B 0,C 180,E1 -1292.589,E2 -1292.589} C_VEL
LIN {X 0,Y 587.169,Z 395.289,A -85,B 0,C 180,E1 -1293.819,E2 -1293.819} C_VEL
LIN {X 0,Y 587.13,Z 399.216,A -85,B 0,C 180,E1 -1295.069,E2 -1295.069} C_VEL
LIN {X 0,Y 587.126,Z 401.077,A -85,B 0,C 180,E1 -1295.912,E2 -1295.912} C_VEL
LIN {X 0,Y 587.123,Z 402.288,A -85,B 0,C 180,E1 -1296.763,E2 -1296.763} C_VEL
LIN {X 0,Y 587.119,Z 402.953,A -85,B 0,C 180,E1 -1297.811,E2 -1297.811} C_VEL
LIN {X 0,Y 587.114,Z 402.659,A -85,B 0,C 180,E1 -1298.915,E2 -1298.915} C_VEL
LIN {X 0,Y 587.145,Z 400.91,A -85,B 0,C 180,E1 -1300.268,E2 -1300.268} C_VEL
LIN {X 0,Y 587.166,Z 397.487,A -85,B 0,C 180,E1 -1301.629,E2 -1301.629} C_VEL
LIN {X 0,Y 587.18,Z 394.19,A -85,B 0,C 180,E1 -1302.551,E2 -1302.551} C_VEL
LIN {X 0,Y 587.182,Z 388.649,A -85,B 0,C 180,E1 -1303.736,E2 -1303.736} C_VEL
LIN {X 0,Y 587.22,Z 381.455,A -85,B 0,C 180,E1 -1304.921,E2 -1304.921} C_VEL
LIN {X 0,Y 587.266,Z 374.014,A -85,B 0,C 180,E1 -1305.893,E2 -1305.893} C_VEL
LIN {X 0,Y 587.347,Z 364.74,A -85,B 0,C 180,E1 -1306.879,E2 -1306.879} C_VEL
LIN {X 0,Y 587.422,Z 355.205,A -85,B 0,C 180,E1 -1307.703,E2 -1307.703} C_VEL
LIN {X 0,Y 587.438,Z 345.39,A -85,B 0,C 180,E1 -1308.395,E2 -1308.395} C_VEL
LIN {X 0,Y 587.522,Z 334.214,A -85,B 0,C 180,E1 -1309.028,E2 -1309.028} C_VEL
LIN {X 0,Y 587.619,Z 322.411,A -85,B 0,C 180,E1 -1309.546,E2 -1309.546} C_VEL
LIN {X 0,Y 587.642,Z 309.637,A -85,B 0,C 180,E1 -1309.959,E2 -1309.959} C_VEL
LIN {X 0,Y 587.734,Z 296.52,A -85,B 0,C 180,E1 -1310.228,E2 -1310.228} C_VEL
LIN {X 0,Y 587.771,Z 196.198,A -85,B 0,C 180,E1 -1311.466,E2 -1311.466} C_VEL
LIN {X 0,Y 587.292,Z 193.373,A -85,B 0,C 180,E1 -1311.518,E2 -1311.518} C_VEL
LIN {X 0,Y 587.33,Z 181.322,A -85,B 0,C 180,E1 -1313.997,E2 -1313.997} C_VEL
LIN {X 0,Y 587.336,Z 181.323,A -85,B 0,C 180,E1 -1316.889,E2 -1316.889} C_VEL
LIN {X 0,Y 587.321,Z 181.326,A -85,B 0,C 180,E1 -1319.493,E2 -1319.493} C_VEL
LIN {X 0,Y 587.342,Z 181.318,A -85,B 0,C 180,E1 -1322.309,E2 -1322.309} C_VEL
LIN {X 0,Y 587.339,Z 181.322,A -85,B 0,C 180,E1 -1325.423,E2 -1325.423} C_VEL
LIN {X 0,Y 587.313,Z 181.321,A -85,B 0,C 180,E1 -1328.225,E2 -1328.225} C_VEL
LIN {X 0,Y 587.341,Z 181.324,A -85,B 0,C 180,E1 -1331.151,E2 -1331.151} C_VEL
LIN {X 0,Y 587.312,Z 181.321,A -85,B 0,C 180,E1 -1334.025,E2 -1334.025} C_VEL
LIN {X 0,Y 587.352,Z 181.317,A -85,B 0,C 180,E1 -1336.154,E2 -1336.154} C_VEL
LIN {X 0,Y 587.339,Z 181.325,A -85,B 0,C 180,E1 -1338.963,E2 -1338.963} C_VEL
LIN {X 0,Y 587.339,Z 181.318,A -85,B 0,C 180,E1 -1341.745,E2 -1341.745} C_VEL
LIN {X 0,Y 587.363,Z 181.323,A -85,B 0,C 180,E1 -1344.507,E2 -1344.507} C_VEL
LIN {X 0,Y 587.354,Z 181.317,A -85,B 0,C 180,E1 -1347.257,E2 -1347.257} C_VEL
LIN {X 0,Y 587.384,Z 181.315,A -85,B 0,C 180,E1 -1350,E2 -1350} C_VEL
LIN {X 0,Y 587.363,Z 181.32,A -85,B 0,C 180,E1 -1352.743,E2 -1352.743} C_VEL
LIN {X 0,Y 587.344,Z 181.317,A -85,B 0,C 180,E1 -1355.493,E2 -1355.493} C_VEL
LIN {X 0,Y 587.363,Z 181.324,A -85,B 0,C 180,E1 -1358.255,E2 -1358.255} C_VEL
LIN {X 0,Y 587.333,Z 181.319,A -85,B 0,C 180,E1 -1361.124,E2 -1361.124} C_VEL
LIN {X 0,Y 587.355,Z 181.32,A -85,B 0,C 180,E1 -1363.846,E2 -1363.846} C_VEL
LIN {X 0,Y 587.323,Z 181.321,A -85,B 0,C 180,E1 -1366.805,E2 -1366.805} C_VEL
LIN {X 0,Y 587.308,Z 181.325,A -85,B 0,C 180,E1 -1369.576,E2 -1369.576} C_VEL
LIN {X 0,Y 587.314,Z 181.327,A -85,B 0,C 180,E1 -1371.775,E2 -1371.775} C_VEL
LIN {X 0,Y 587.314,Z 181.321,A -85,B 0,C 180,E1 -1374.76,E2 -1374.76} C_VEL
LIN {X 0,Y 587.306,Z 181.329,A -85,B 0,C 180,E1 -1377.684,E2 -1377.684} C_VEL
LIN {X 0,Y 587.317,Z 181.324,A -85,B 0,C 180,E1 -1380.171,E2 -1380.171} C_VEL
LIN {X 0,Y 587.33,Z 181.319,A -85,B 0,C 180,E1 -1382.58,E2 -1382.58} C_VEL
LIN {X 0,Y 587.321,Z 181.322,A -85,B 0,C 180,E1 -1385.056,E2 -1385.056} C_VEL
LIN {X 0,Y 587.332,Z 181.325,A -85,B 0,C 180,E1 -1387.837,E2 -1387.837} C_VEL
LIN {X 0,Y 587.307,Z 181.323,A -85,B 0,C 180,E1 -1390.255,E2 -1390.255} C_VEL
LIN {X 0,Y 587.303,Z 181.326,A -85,B 0,C 180,E1 -1393.117,E2 -1393.117} C_VEL
LIN {X 0,Y 587.3,Z 181.324,A -85,B 0,C 180,E1 -1396.047,E2 -1396.047} C_VEL
LIN {X 0,Y 587.333,Z 181.322,A -85,B 0,C 180,E1 -1398.926,E2 -1398.926} C_VEL
LIN {X 0,Y 587.318,Z 181.326,A -85,B 0,C 180,E1 -1401.52,E2 -1401.52} C_VEL
LIN {X 0,Y 587.288,Z 181.324,A -85,B 0,C 180,E1 -1404.1,E2 -1404.1} C_VEL
LIN {X 0,Y 587.336,Z 181.324,A -85,B 0,C 180,E1 -1406.889,E2 -1406.889} C_VEL
LIN {X 0,Y 587.322,Z 181.324,A -85,B 0,C 180,E1 -1409.493,E2 -1409.493} C_VEL
LIN {X 0,Y 587.297,Z 181.323,A -85,B 0,C 180,E1 -1412.18,E2 -1412.18} C_VEL
LIN {X 0,Y 587.325,Z 181.322,A -85,B 0,C 180,E1 -1414.483,E2 -1414.483} C_VEL
LIN {X 0,Y 587.31,Z 181.323,A -85,B 0,C 180,E1 -1417.485,E2 -1417.485} C_VEL
LIN {X 0,Y 587.312,Z 181.321,A -85,B 0,C 180,E1 -1419.695,E2 -1419.695} C_VEL
LIN {X 0,Y 587.284,Z 181.325,A -85,B 0,C 180,E1 -1421.872,E2 -1421.872} C_VEL
LIN {X 0,Y 587.302,Z 181.323,A -85,B 0,C 180,E1 -1424.024,E2 -1424.024} C_VEL
LIN {X 0,Y 587.342,Z 181.32,A -85,B 0,C 180,E1 -1426.154,E2 -1426.154} C_VEL
LIN {X 0,Y 587.341,Z 181.322,A -85,B 0,C 180,E1 -1428.962,E2 -1428.962} C_VEL
LIN {X 0,Y 587.336,Z 181.318,A -85,B 0,C 180,E1 -1431.744,E2 -1431.744} C_VEL
LIN {X 0,Y 587.349,Z 181.327,A -85,B 0,C 180,E1 -1434.507,E2 -1434.507} C_VEL
LIN {X 0,Y 587.348,Z 181.317,A -85,B 0,C 180,E1 -1437.257,E2 -1437.257} C_VEL
LIN {X 0,Y 587.384,Z 181.316,A -85,B 0,C 180,E1 -1440,E2 -1440} C_VEL
LIN {X 0,Y 587.353,Z 181.319,A -85,B 0,C 180,E1 -1442.743,E2 -1442.743} C_VEL
LIN {X 0,Y 587.341,Z 181.318,A -85,B 0,C 180,E1 -1445.493,E2 -1445.493} C_VEL
LIN {X 0,Y 587.339,Z 181.326,A -85,B 0,C 180,E1 -1448.256,E2 -1448.256} C_VEL
LIN {X 0,Y 587.334,Z 181.318,A -85,B 0,C 180,E1 -1451.124,E2 -1451.124} C_VEL
LIN {X 0,Y 587.343,Z 181.324,A -85,B 0,C 180,E1 -1454.25,E2 -1454.25} C_VEL
LIN {X 0,Y 587.287,Z 181.324,A -85,B 0,C 180,E1 -1456.793,E2 -1456.793} C_VEL
LIN {X 0,Y 587.304,Z 181.327,A -85,B 0,C 180,E1 -1459.577,E2 -1459.577} C_VEL
LIN {X 0,Y 587.311,Z 181.33,A -85,B 0,C 180,E1 -1461.775,E2 -1461.775} C_VEL
LIN {X 0,Y 587.303,Z 181.322,A -85,B 0,C 180,E1 -1464.761,E2 -1464.761} C_VEL
LIN {X 0,Y 587.301,Z 181.333,A -85,B 0,C 180,E1 -1467.683,E2 -1467.683} C_VEL
LIN {X 0,Y 587.314,Z 181.323,A -85,B 0,C 180,E1 -1470.171,E2 -1470.171} C_VEL
LIN {X 0,Y 587.327,Z 181.319,A -85,B 0,C 180,E1 -1472.58,E2 -1472.58} C_VEL
LIN {X 0,Y 587.305,Z 181.325,A -85,B 0,C 180,E1 -1475.057,E2 -1475.057} C_VEL
LIN {X 0,Y 587.328,Z 181.323,A -85,B 0,C 180,E1 -1477.837,E2 -1477.837} C_VEL
LIN {X 0,Y 587.305,Z 181.322,A -85,B 0,C 180,E1 -1480.255,E2 -1480.255} C_VEL
LIN {X 0,Y 587.292,Z 181.33,A -85,B 0,C 180,E1 -1483.115,E2 -1483.115} C_VEL
LIN {X 0,Y 587.3,Z 181.323,A -85,B 0,C 180,E1 -1486.047,E2 -1486.047} C_VEL
LIN {X 0,Y 587.333,Z 181.324,A -85,B 0,C 180,E1 -1488.926,E2 -1488.926} C_VEL
LIN {X 0,Y 587.314,Z 181.325,A -85,B 0,C 180,E1 -1491.519,E2 -1491.519} C_VEL
LIN {X 0,Y 587.278,Z 181.325,A -85,B 0,C 180,E1 -1494.099,E2 -1494.099} C_VEL
LIN {X 0,Y 587.334,Z 181.327,A -85,B 0,C 180,E1 -1496.889,E2 -1496.889} C_VEL
LIN {X 0,Y 587.308,Z 181.324,A -85,B 0,C 180,E1 -1499.495,E2 -1499.495} C_VEL
LIN {X 0,Y 587.291,Z 181.327,A -85,B 0,C 180,E1 -1501.401,E2 -1501.401} C_VEL
LIN {X 0,Y 587.307,Z 181.323,A -85,B 0,C 180,E1 -1503.83,E2 -1503.83} C_VEL
LIN {X 0,Y 587.343,Z 181.498,A -85,B 0,C 180,E1 -1505.338,E2 -1505.338} C_VEL
LIN {X 0,Y 588.034,Z 185.418,A -85,B 0,C 180,E1 -1505.86,E2 -1505.86} C_VEL
LIN {X 0,Y 587.876,Z 207.165,A -85,B 0,C 180,E1 -1508.639,E2 -1508.639} C_VEL
LIN {X 0,Y 587.704,Z 228.507,A -85,B 0,C 180,E1 -1511.344,E2 -1511.344} C_VEL
LIN {X 0,Y 587.577,Z 251.468,A -85,B 0,C 180,E1 -1514.21,E2 -1514.21} C_VEL
LIN {X 0,Y 587.413,Z 269.944,A -85,B 0,C 180,E1 -1516.486,E2 -1516.486} C_VEL
LIN {X 0,Y 587.854,Z 274.701,A -85,B 0,C 180,E1 -1516.562,E2 -1516.562} C_VEL
LIN {X 0,Y 587.75,Z 378.935,A -85,B 0,C 180,E1 -1517.855,E2 -1517.855} C_VEL
LIN {X 0,Y 587.67,Z 392.211,A -85,B 0,C 180,E1 -1518.16,E2 -1518.16} C_VEL
LIN {X 0,Y 587.613,Z 404.641,A -85,B 0,C 180,E1 -1518.585,E2 -1518.585} C_VEL
LIN {X 0,Y 587.557,Z 416.626,A -85,B 0,C 180,E1 -1519.141,E2 -1519.141} C_VEL
LIN {X 0,Y 587.464,Z 428.199,A -85,B 0,C 180,E1 -1519.836,E2 -1519.836} C_VEL
LIN {X 0,Y 587.366,Z 438.596,A -85,B 0,C 180,E1 -1520.617,E2 -1520.617} C_VEL
LIN {X 0,Y 587.322,Z 447.11,A -85,B 0,C 180,E1 -1521.397,E2 -1521.397} C_VEL
LIN {X 0,Y 587.274,Z 454.959,A -85,B 0,C 180,E1 -1522.263,E2 -1522.263} C_VEL
LIN {X 0,Y 587.23,Z 461.468,A -85,B 0,C 180,E1 -1523.126,E2 -1523.126} C_VEL
LIN {X 0,Y 587.237,Z 467.865,A -85,B 0,C 180,E1 -1524.161,E2 -1524.161} C_VEL
LIN {X 0,Y 587.147,Z 472.949,A -85,B 0,C 180,E1 -1525.193,E2 -1525.193} C_VEL
LIN {X 0,Y 587.213,Z 476.895,A -85,B 0,C 180,E1 -1526.226,E2 -1526.226} C_VEL
LIN {X 0,Y 587.132,Z 479.808,A -85,B 0,C 180,E1 -1527.255,E2 -1527.255} C_VEL
LIN {X 0,Y 587.141,Z 481.199,A -85,B 0,C 180,E1 -1527.942,E2 -1527.942} C_VEL
LIN {X 0,Y 587.14,Z 482.784,A -85,B 0,C 180,E1 -1529.314,E2 -1529.314} C_VEL
LIN {X 0,Y 587.137,Z 483,A -85,B 0,C 180,E1 -1530,E2 -1530} C_VEL
LIN {X 0,Y 587.147,Z 482.186,A -85,B 0,C 180,E1 -1531.372,E2 -1531.372} C_VEL
LIN {X 0,Y 587.141,Z 481.201,A -85,B 0,C 180,E1 -1532.058,E2 -1532.058} C_VEL
LIN {X 0,Y 587.132,Z 479.81,A -85,B 0,C 180,E1 -1532.744,E2 -1532.744} C_VEL
LIN {X 0,Y 587.213,Z 476.896,A -85,B 0,C 180,E1 -1533.774,E2 -1533.774} C_VEL
LIN {X 0,Y 587.147,Z 472.95,A -85,B 0,C 180,E1 -1534.806,E2 -1534.806} C_VEL
LIN {X 0,Y 587.218,Z 466.878,A -85,B 0,C 180,E1 -1536.011,E2 -1536.011} C_VEL
LIN {X 0,Y 587.245,Z 460.238,A -85,B 0,C 180,E1 -1537.046,E2 -1537.046} C_VEL
LIN {X 0,Y 587.299,Z 451.992,A -85,B 0,C 180,E1 -1538.083,E2 -1538.083} C_VEL
LIN {X 0,Y 587.343,Z 443.54,A -85,B 0,C 180,E1 -1538.949,E2 -1538.949} C_VEL
LIN {X 0,Y 587.419,Z 433.098,A -85,B 0,C 180,E1 -1539.816,E2 -1539.816} C_VEL
LIN {X 0,Y 587.497,Z 422.759,A -85,B 0,C 180,E1 -1540.511,E2 -1540.511} C_VEL
LIN {X 0,Y 587.561,Z 410.82,A -85,B 0,C 180,E1 -1541.149,E2 -1541.149} C_VEL
LIN {X 0,Y 587.629,Z 398.603,A -85,B 0,C 180,E1 -1541.639,E2 -1541.639} C_VEL
LIN {X 0,Y 587.705,Z 385.442,A -85,B 0,C 180,E1 -1542.014,E2 -1542.014} C_VEL
LIN {X 0,Y 587.768,Z 373.096,A -85,B 0,C 180,E1 -1542.231,E2 -1542.231} C_VEL
LIN {X 0,Y 587.737,Z 272.274,A -85,B 0,C 180,E1 -1543.47,E2 -1543.47} C_VEL
LIN {X 0,Y 587.418,Z 269.768,A -85,B 0,C 180,E1 -1543.535,E2 -1543.535} C_VEL
LIN {X 0,Y 587.56,Z 245.731,A -85,B 0,C 180,E1 -1546.504,E2 -1546.504} C_VEL
LIN {X 0,Y 587.729,Z 224.606,A -85,B 0,C 180,E1 -1549.148,E2 -1549.148} C_VEL
LIN {X 0,Y 587.909,Z 204.115,A -85,B 0,C 180,E1 -1551.751,E2 -1551.751} C_VEL
LIN {X 0,Y 587.998,Z 185.325,A -85,B 0,C 180,E1 -1554.141,E2 -1554.141} C_VEL
LIN {X 0,Y 587.302,Z 181.33,A -85,B 0,C 180,E1 -1554.663,E2 -1554.663} C_VEL
LIN {X 0,Y 587.326,Z 181.329,A -85,B 0,C 180,E1 -1557.046,E2 -1557.046} C_VEL
LIN {X 0,Y 587.305,Z 181.328,A -85,B 0,C 180,E1 -1559.382,E2 -1559.382} C_VEL
LIN {X 0,Y 587.315,Z 181.322,A -85,B 0,C 180,E1 -1561.83,E2 -1561.83} C_VEL
LIN {X 0,Y 587.332,Z 181.321,A -85,B 0,C 180,E1 -1564.345,E2 -1564.345} C_VEL
LIN {X 0,Y 587.338,Z 181.319,A -85,B 0,C 180,E1 -1567.608,E2 -1567.608} C_VEL
LIN {X 0,Y 587.302,Z 181.325,A -85,B 0,C 180,E1 -1570.255,E2 -1570.255} C_VEL
LIN {X 0,Y 587.304,Z 181.327,A -85,B 0,C 180,E1 -1573.007,E2 -1573.007} C_VEL
LIN {X 0,Y 587.312,Z 181.323,A -85,B 0,C 180,E1 -1576.048,E2 -1576.048} C_VEL
LIN {X 0,Y 587.335,Z 181.322,A -85,B 0,C 180,E1 -1578.925,E2 -1578.925} C_VEL
LIN {X 0,Y 587.316,Z 181.321,A -85,B 0,C 180,E1 -1581.519,E2 -1581.519} C_VEL
LIN {X 0,Y 587.287,Z 181.33,A -85,B 0,C 180,E1 -1584.099,E2 -1584.099} C_VEL
LIN {X 0,Y 587.336,Z 181.32,A -85,B 0,C 180,E1 -1586.889,E2 -1586.889} C_VEL
LIN {X 0,Y 587.32,Z 181.321,A -85,B 0,C 180,E1 -1589.493,E2 -1589.493} C_VEL
LIN {X 0,Y 587.341,Z 181.324,A -85,B 0,C 180,E1 -1592.309,E2 -1592.309} C_VEL
LIN {X 0,Y 587.34,Z 181.319,A -85,B 0,C 180,E1 -1595.423,E2 -1595.423} C_VEL
LIN {X 0,Y 587.315,Z 181.327,A -85,B 0,C 180,E1 -1598.225,E2 -1598.225} C_VEL
LIN {X 0,Y 587.333,Z 181.32,A -85,B 0,C 180,E1 -1601.151,E2 -1601.151} C_VEL
LIN {X 0,Y 587.309,Z 181.328,A -85,B 0,C 180,E1 -1604.024,E2 -1604.024} C_VEL
LIN {X 0,Y 587.354,Z 181.32,A -85,B 0,C 180,E1 -1606.154,E2 -1606.154} C_VEL
LIN {X 0,Y 587.337,Z 181.319,A -85,B 0,C 180,E1 -1608.962,E2 -1608.962} C_VEL
LIN {X 0,Y 587.364,Z 181.322,A -85,B 0,C 180,E1 -1611.745,E2 -1611.745} C_VEL
LIN {X 0,Y 587.35,Z 181.317,A -85,B 0,C 180,E1 -1614.507,E2 -1614.507} C_VEL
LIN {X 0,Y 587.375,Z 181.321,A -85,B 0,C 180,E1 -1617.257,E2 -1617.257} C_VEL
LIN {X 0,Y 587.383,Z 181.314,A -85,B 0,C 180,E1 -1620,E2 -1620} C_VEL
LIN {X 0,Y 587.36,Z 181.318,A -85,B 0,C 180,E1 -1622.743,E2 -1622.743} C_VEL
LIN {X 0,Y 587.367,Z 181.32,A -85,B 0,C 180,E1 -1625.493,E2 -1625.493} C_VEL
LIN {X 0,Y 587.341,Z 181.318,A -85,B 0,C 180,E1 -1628.256,E2 -1628.256} C_VEL
LIN {X 0,Y 587.349,Z 181.326,A -85,B 0,C 180,E1 -1631.134,E2 -1631.134} C_VEL
LIN {X 0,Y 587.365,Z 181.317,A -85,B 0,C 180,E1 -1634.26,E2 -1634.26} C_VEL
LIN {X 0,Y 587.343,Z 181.32,A -85,B 0,C 180,E1 -1637.406,E2 -1637.406} C_VEL
LIN {X 0,Y 587.301,Z 181.325,A -85,B 0,C 180,E1 -1638.292,E2 -1638.292} C_VEL
LIN {X 0,Y 586.66,Z 181.413,A -85,B 0,C 180,E1 -1638.864,E2 -1638.864} C_VEL
LIN {X 0,Y 583.837,Z 181.765,A -85,B 0,C 180,E1 -1639.792,E2 -1639.792} C_VEL
LIN {X 0,Y 581.43,Z 182.063,A -85,B 0,C 180,E1 -1640.539,E2 -1640.539} C_VEL
LIN {X 0,Y 580.382,Z 182.191,A -85,B 0,C 180,E1 -1641.116,E2 -1641.116} C_VEL
LIN {X 0,Y 580.29,Z 182.2,A -85,B 0,C 180,E1 -1641.311,E2 -1641.311} C_VEL
LIN {X 0,Y 580.285,Z 182.376,A -85,B 0,C 180,E1 -1642.146,E2 -1642.146} C_VEL
LIN {X 0,Y 580.264,Z 193.37,A -85,B 0,C 180,E1 -1644.405,E2 -1644.405} C_VEL
LIN {X 0,Y 580.98,Z 199.426,A -85,B 0,C 180,E1 -1644.504,E2 -1644.504} C_VEL
LIN {X 0,Y 580.778,Z 299.62,A -85,B 0,C 180,E1 -1645.766,E2 -1645.766} C_VEL
LIN {X 0,Y 580.706,Z 313.423,A -85,B 0,C 180,E1 -1646.097,E2 -1646.097} C_VEL
LIN {X 0,Y 580.645,Z 325.695,A -85,B 0,C 180,E1 -1646.534,E2 -1646.534} C_VEL
LIN {X 0,Y 580.507,Z 337.442,A -85,B 0,C 180,E1 -1647.098,E2 -1647.098} C_VEL
LIN {X 0,Y 580.412,Z 348.954,A -85,B 0,C 180,E1 -1647.808,E2 -1647.808} C_VEL
LIN {X 0,Y 580.358,Z 358.947,A -85,B 0,C 180,E1 -1648.577,E2 -1648.577} C_VEL
LIN {X 0,Y 580.291,Z 368.73,A -85,B 0,C 180,E1 -1649.507,E2 -1649.507} C_VEL
LIN {X 0,Y 580.186,Z 377.833,A -85,B 0,C 180,E1 -1650.581,E2 -1650.581} C_VEL
LIN {X 0,Y 580.162,Z 385.365,A -85,B 0,C 180,E1 -1651.699,E2 -1651.699} C_VEL
LIN {X 0,Y 580.087,Z 390.405,A -85,B 0,C 180,E1 -1652.625,E2 -1652.625} C_VEL
LIN {X 0,Y 580.081,Z 395.656,A -85,B 0,C 180,E1 -1653.87,E2 -1653.87} C_VEL
LIN {X 0,Y 580.044,Z 399.481,A -85,B 0,C 180,E1 -1655.136,E2 -1655.136} C_VEL
LIN {X 0,Y 580.015,Z 401.916,A -85,B 0,C 180,E1 -1656.422,E2 -1656.422} C_VEL
LIN {X 0,Y 580.026,Z 402.744,A -85,B 0,C 180,E1 -1657.289,E2 -1657.289} C_VEL
LIN {X 0,Y 580.016,Z 402.979,A -85,B 0,C 180,E1 -1658.168,E2 -1658.168} C_VEL
LIN {X 0,Y 580.02,Z 402.496,A -85,B 0,C 180,E1 -1659.152,E2 -1659.152} C_VEL
LIN {X 0,Y 580.044,Z 401.012,A -85,B 0,C 180,E1 -1660.242,E2 -1660.242} C_VEL
LIN {X 0,Y 580.042,Z 398.581,A -85,B 0,C 180,E1 -1661.305,E2 -1661.305} C_VEL
LIN {X 0,Y 580.092,Z 395.188,A -85,B 0,C 180,E1 -1662.351,E2 -1662.351} C_VEL
LIN {X 0,Y 580.108,Z 390.834,A -85,B 0,C 180,E1 -1663.373,E2 -1663.373} C_VEL
LIN {X 0,Y 580.155,Z 385.432,A -85,B 0,C 180,E1 -1664.379,E2 -1664.379} C_VEL
LIN {X 0,Y 580.183,Z 378.905,A -85,B 0,C 180,E1 -1665.366,E2 -1665.366} C_VEL
LIN {X 0,Y 580.228,Z 371.016,A -85,B 0,C 180,E1 -1666.337,E2 -1666.337} C_VEL
LIN {X 0,Y 580.301,Z 361.414,A -85,B 0,C 180,E1 -1667.296,E2 -1667.296} C_VEL
LIN {X 0,Y 580.437,Z 351.108,A -85,B 0,C 180,E1 -1668.13,E2 -1668.13} C_VEL
LIN {X 0,Y 580.455,Z 340.198,A -85,B 0,C 180,E1 -1668.838,E2 -1668.838} C_VEL
LIN {X 0,Y 580.624,Z 327.699,A -85,B 0,C 180,E1 -1669.469,E2 -1669.469} C_VEL
LIN {X 0,Y 580.722,Z 315.337,A -85,B 0,C 180,E1 -1669.936,E2 -1669.936} C_VEL
LIN {X 0,Y 580.781,Z 302.682,A -85,B 0,C 180,E1 -1670.265,E2 -1670.265} C_VEL
LIN {X 0,Y 580.851,Z 285.673,A -85,B 0,C 180,E1 -1670.517,E2 -1670.517} C_VEL
LIN {X 0,Y 580.846,Z 196.837,A -85,B 0,C 180,E1 -1671.621,E2 -1671.621} C_VEL
LIN {X 0,Y 580.242,Z 193.373,A -85,B 0,C 180,E1 -1671.685,E2 -1671.685} C_VEL
LIN {X 0,Y 580.295,Z 182.199,A -85,B 0,C 180,E1 -1673.992,E2 -1673.992} C_VEL
LIN {X 0,Y 580.288,Z 182.202,A -85,B 0,C 180,E1 -1676.975,E2 -1676.975} C_VEL
LIN {X 0,Y 580.283,Z 182.204,A -85,B 0,C 180,E1 -1679.424,E2 -1679.424} C_VEL
LIN {X 0,Y 580.29,Z 182.196,A -85,B 0,C 180,E1 -1682.143,E2 -1682.143} C_VEL
LIN {X 0,Y 580.287,Z 182.203,A -85,B 0,C 180,E1 -1684.92,E2 -1684.92} C_VEL
LIN {X 0,Y 580.255,Z 182.2,A -85,B 0,C 180,E1 -1687.947,E2 -1687.947} C_VEL
LIN {X 0,Y 580.294,Z 182.205,A -85,B 0,C 180,E1 -1690.913,E2 -1690.913} C_VEL
LIN {X 0,Y 580.262,Z 182.199,A -85,B 0,C 180,E1 -1693.825,E2 -1693.825} C_VEL
LIN {X 0,Y 580.266,Z 182.207,A -85,B 0,C 180,E1 -1696.696,E2 -1696.696} C_VEL
LIN {X 0,Y 580.307,Z 182.203,A -85,B 0,C 180,E1 -1698.827,E2 -1698.827} C_VEL
LIN {X 0,Y 580.308,Z 182.194,A -85,B 0,C 180,E1 -1701.644,E2 -1701.644} C_VEL
LIN {X 0,Y 580.329,Z 182.198,A -85,B 0,C 180,E1 -1704.44,E2 -1704.44} C_VEL
LIN {X 0,Y 580.342,Z 182.191,A -85,B 0,C 180,E1 -1707.918,E2 -1707.918} C_VEL
LIN {X 0,Y 580.358,Z 182.194,A -85,B 0,C 180,E1 -1710.694,E2 -1710.694} C_VEL
LIN {X 0,Y 580.328,Z 182.196,A -85,B 0,C 180,E1 -1712.777,E2 -1712.777} C_VEL
LIN {X 0,Y 580.313,Z 182.193,A -85,B 0,C 180,E1 -1715.56,E2 -1715.56} C_VEL
LIN {X 0,Y 580.326,Z 182.201,A -85,B 0,C 180,E1 -1718.356,E2 -1718.356} C_VEL
LIN {X 0,Y 580.303,Z 182.194,A -85,B 0,C 180,E1 -1721.191,E2 -1721.191} C_VEL
LIN {X 0,Y 580.314,Z 182.2,A -85,B 0,C 180,E1 -1724.017,E2 -1724.017} C_VEL
LIN {X 0,Y 580.292,Z 182.196,A -85,B 0,C 180,E1 -1726.906,E2 -1726.906} C_VEL
LIN {X 0,Y 580.282,Z 182.203,A -85,B 0,C 180,E1 -1729.823,E2 -1729.823} C_VEL
LIN {X 0,Y 580.257,Z 182.209,A -85,B 0,C 180,E1 -1732.053,E2 -1732.053} C_VEL
LIN {X 0,Y 580.289,Z 182.196,A -85,B 0,C 180,E1 -1735.081,E2 -1735.081} C_VEL
LIN {X 0,Y 580.277,Z 182.202,A -85,B 0,C 180,E1 -1738.187,E2 -1738.187} C_VEL
LIN {X 0,Y 580.272,Z 182.198,A -85,B 0,C 180,E1 -1740.692,E2 -1740.692} C_VEL
LIN {X 0,Y 580.303,Z 182.198,A -85,B 0,C 180,E1 -1743.316,E2 -1743.316} C_VEL
LIN {X 0,Y 580.244,Z 182.21,A -85,B 0,C 180,E1 -1745.756,E2 -1745.756} C_VEL
LIN {X 0,Y 580.284,Z 182.199,A -85,B 0,C 180,E1 -1748.147,E2 -1748.147} C_VEL
LIN {X 0,Y 580.297,Z 182.196,A -85,B 0,C 180,E1 -1750.844,E2 -1750.844} C_VEL
LIN {X 0,Y 580.271,Z 182.205,A -85,B 0,C 180,E1 -1753.659,E2 -1753.659} C_VEL
LIN {X 0,Y 580.245,Z 182.202,A -85,B 0,C 180,E1 -1756.613,E2 -1756.613} C_VEL
LIN {X 0,Y 580.295,Z 182.202,A -85,B 0,C 180,E1 -1759.156,E2 -1759.156} C_VEL
LIN {X 0,Y 580.286,Z 182.198,A -85,B 0,C 180,E1 -1761.928,E2 -1761.928} C_VEL
LIN {X 0,Y 580.25,Z 182.201,A -85,B 0,C 180,E1 -1764.453,E2 -1764.453} C_VEL
LIN {X 0,Y 580.287,Z 182.203,A -85,B 0,C 180,E1 -1766.975,E2 -1766.975} C_VEL
LIN {X 0,Y 580.283,Z 182.201,A -85,B 0,C 180,E1 -1769.424,E2 -1769.424} C_VEL
LIN {X 0,Y 580.25,Z 182.201,A -85,B 0,C 180,E1 -1772.151,E2 -1772.151} C_VEL
LIN {X 0,Y 580.283,Z 182.206,A -85,B 0,C 180,E1 -1774.919,E2 -1774.919} C_VEL
LIN {X 0,Y 580.255,Z 182.2,A -85,B 0,C 180,E1 -1777.947,E2 -1777.947} C_VEL
LIN {X 0,Y 580.3,Z 182.204,A -85,B 0,C 180,E1 -1780.85,E2 -1780.85} C_VEL
LIN {X 0,Y 580.253,Z 182.2,A -85,B 0,C 180,E1 -1783.825,E2 -1783.825} C_VEL
LIN {X 0,Y 580.299,Z 182.196,A -85,B 0,C 180,E1 -1785.982,E2 -1785.982} C_VEL
LIN {X 0,Y 580.31,Z 182.2,A -85,B 0,C 180,E1 -1788.827,E2 -1788.827} C_VEL
LIN {X 0,Y 580.305,Z 182.194,A -85,B 0,C 180,E1 -1791.644,E2 -1791.644} C_VEL
LIN {X 0,Y 580.315,Z 182.202,A -85,B 0,C 180,E1 -1794.44,E2 -1794.44} C_VEL
LIN {X 0,Y 580.341,Z 182.192,A -85,B 0,C 180,E1 -1797.918,E2 -1797.918} C_VEL
LIN {X 0,Y 580.35,Z 182.193,A -85,B 0,C 180,E1 -1800.694,E2 -1800.694} C_VEL
LIN {X 0,Y 580.319,Z 182.195,A -85,B 0,C 180,E1 -1802.777,E2 -1802.777} C_VEL
LIN {X 0,Y 580.311,Z 182.194,A -85,B 0,C 180,E1 -1805.56,E2 -1805.56} C_VEL
LIN {X 0,Y 580.307,Z 182.201,A -85,B 0,C 180,E1 -1808.356,E2 -1808.356} C_VEL
LIN {X 0,Y 580.305,Z 182.194,A -85,B 0,C 180,E1 -1811.191,E2 -1811.191} C_VEL
LIN {X 0,Y 580.301,Z 182.2,A -85,B 0,C 180,E1 -1814.331,E2 -1814.331} C_VEL
LIN {X 0,Y 580.253,Z 182.2,A -85,B 0,C 180,E1 -1816.899,E2 -1816.899} C_VEL
LIN {X 0,Y 580.277,Z 182.206,A -85,B 0,C 180,E1 -1819.823,E2 -1819.823} C_VEL
LIN {X 0,Y 580.281,Z 182.197,A -85,B 0,C 180,E1 -1822.803,E2 -1822.803} C_VEL
LIN {X 0,Y 580.265,Z 182.207,A -85,B 0,C 180,E1 -1825.85,E2 -1825.85} C_VEL
LIN {X 0,Y 580.281,Z 182.198,A -85,B 0,C 180,E1 -1828.977,E2 -1828.977} C_VEL
LIN {X 0,Y 580.269,Z 182.205,A -85,B 0,C 180,E1 -1831.386,E2 -1831.386} C_VEL
LIN {X 0,Y 580.276,Z 182.203,A -85,B 0,C 180,E1 -1833.858,E2 -1833.858} C_VEL
LIN {X 0,Y 580.278,Z 182.199,A -85,B 0,C 180,E1 -1836.931,E2 -1836.931} C_VEL
LIN {X 0,Y 580.276,Z 182.2,A -85,B 0,C 180,E1 -1839.934,E2 -1839.934} C_VEL
LIN {X 0,Y 580.254,Z 182.202,A -85,B 0,C 180,E1 -1842.709,E2 -1842.709} C_VEL
LIN {X 0,Y 580.253,Z 182.205,A -85,B 0,C 180,E1 -1845.611,E2 -1845.611} C_VEL
LIN {X 0,Y 580.271,Z 182.2,A -85,B 0,C 180,E1 -1848.67,E2 -1848.67} C_VEL
LIN {X 0,Y 580.267,Z 182.206,A -85,B 0,C 180,E1 -1850.964,E2 -1850.964} C_VEL
LIN {X 0,Y 580.246,Z 182.204,A -85,B 0,C 180,E1 -1853.594,E2 -1853.594} C_VEL
LIN {X 0,Y 580.274,Z 182.198,A -85,B 0,C 180,E1 -1856.142,E2 -1856.142} C_VEL
LIN {X 0,Y 580.266,Z 182.204,A -85,B 0,C 180,E1 -1858.614,E2 -1858.614} C_VEL
LIN {X 0,Y 580.278,Z 182.207,A -85,B 0,C 180,E1 -1861.023,E2 -1861.023} C_VEL
LIN {X 0,Y 580.266,Z 182.201,A -85,B 0,C 180,E1 -1863.672,E2 -1863.672} C_VEL
LIN {X 0,Y 580.295,Z 182.403,A -85,B 0,C 180,E1 -1865.192,E2 -1865.192} C_VEL
LIN {X 0,Y 581.07,Z 186.247,A -85,B 0,C 180,E1 -1865.718,E2 -1865.718} C_VEL
LIN {X 0,Y 580.963,Z 207.252,A -85,B 0,C 180,E1 -1868.385,E2 -1868.385} C_VEL
LIN {X 0,Y 580.772,Z 227.072,A -85,B 0,C 180,E1 -1870.929,E2 -1870.929} C_VEL
LIN {X 0,Y 580.595,Z 250.033,A -85,B 0,C 180,E1 -1873.834,E2 -1873.834} C_VEL
LIN {X 0,Y 580.441,Z 270.229,A -85,B 0,C 180,E1 -1876.332,E2 -1876.332} C_VEL
LIN {X 0,Y 580.944,Z 274.701,A -85,B 0,C 180,E1 -1876.4,E2 -1876.4} C_VEL
LIN {X 0,Y 580.827,Z 378.935,A -85,B 0,C 180,E1 -1877.708,E2 -1877.708} C_VEL
LIN {X 0,Y 580.725,Z 392.211,A -85,B 0,C 180,E1 -1878.016,E2 -1878.016} C_VEL
LIN {X 0,Y 580.646,Z 405.146,A -85,B 0,C 180,E1 -1878.466,E2 -1878.466} C_VEL
LIN {X 0,Y 580.579,Z 416.624,A -85,B 0,C 180,E1 -1879.009,E2 -1879.009} C_VEL
LIN {X 0,Y 580.441,Z 428.199,A -85,B 0,C 180,E1 -1879.712,E2 -1879.712} C_VEL
LIN {X 0,Y 580.345,Z 438.598,A -85,B 0,C 180,E1 -1880.503,E2 -1880.503} C_VEL
LIN {X 0,Y 580.271,Z 447.11,A -85,B 0,C 180,E1 -1881.292,E2 -1881.292} C_VEL
LIN {X 0,Y 580.222,Z 454.959,A -85,B 0,C 180,E1 -1882.168,E2 -1882.168} C_VEL
LIN {X 0,Y 580.154,Z 462.65,A -85,B 0,C 180,E1 -1883.221,E2 -1883.221} C_VEL
LIN {X 0,Y 580.139,Z 469.679,A -85,B 0,C 180,E1 -1884.438,E2 -1884.438} C_VEL
LIN {X 0,Y 580.108,Z 474.371,A -85,B 0,C 180,E1 -1885.483,E2 -1885.483} C_VEL
LIN {X 0,Y 580.123,Z 477.957,A -85,B 0,C 180,E1 -1886.527,E2 -1886.527} C_VEL
LIN {X 0,Y 580.043,Z 479.808,A -85,B 0,C 180,E1 -1887.222,E2 -1887.222} C_VEL
LIN {X 0,Y 580.04,Z 481.198,A -85,B 0,C 180,E1 -1887.917,E2 -1887.917} C_VEL
LIN {X 0,Y 580.04,Z 482.785,A -85,B 0,C 180,E1 -1889.306,E2 -1889.306} C_VEL
LIN {X 0,Y 580.037,Z 483,A -85,B 0,C 180,E1 -1890,E2 -1890} C_VEL
LIN {X 0,Y 580.047,Z 482.186,A -85,B 0,C 180,E1 -1891.388,E2 -1891.388} C_VEL
LIN {X 0,Y 580.04,Z 481.2,A -85,B 0,C 180,E1 -1892.083,E2 -1892.083} C_VEL
LIN {X 0,Y 580.043,Z 479.81,A -85,B 0,C 180,E1 -1892.778,E2 -1892.778} C_VEL
LIN {X 0,Y 580.11,Z 476.896,A -85,B 0,C 180,E1 -1893.82,E2 -1893.82} C_VEL
LIN {X 0,Y 580.053,Z 472.95,A -85,B 0,C 180,E1 -1894.865,E2 -1894.865} C_VEL
LIN {X 0,Y 580.139,Z 466.878,A -85,B 0,C 180,E1 -1896.085,E2 -1896.085} C_VEL
LIN {X 0,Y 580.184,Z 460.239,A -85,B 0,C 180,E1 -1897.132,E2 -1897.132} C_VEL
LIN {X 0,Y 580.25,Z 451.992,A -85,B 0,C 180,E1 -1898.182,E2 -1898.182} C_VEL
LIN {X 0,Y 580.308,Z 443.54,A -85,B 0,C 180,E1 -1899.058,E2 -1899.058} C_VEL
LIN {X 0,Y 580.422,Z 433.1,A -85,B 0,C 180,E1 -1899.936,E2 -1899.936} C_VEL
LIN {X 0,Y 580.506,Z 422.758,A -85,B 0,C 180,E1 -1900.639,E2 -1900.639} C_VEL
LIN {X 0,Y 580.596,Z 411.249,A -85,B 0,C 180,E1 -1901.264,E2 -1901.264} C_VEL
LIN {X 0,Y 580.681,Z 398.476,A -85,B 0,C 180,E1 -1901.785,E2 -1901.785} C_VEL
LIN {X 0,Y 580.778,Z 385.44,A -85,B 0,C 180,E1 -1902.159,E2 -1902.159} C_VEL
LIN {X 0,Y 580.844,Z 373.096,A -85,B 0,C 180,E1 -1902.38,E2 -1902.38} C_VEL
LIN {X 0,Y 580.772,Z 272.395,A -85,B 0,C 180,E1 -1903.633,E2 -1903.633} C_VEL
LIN {X 0,Y 580.443,Z 269.947,A -85,B 0,C 180,E1 -1903.679,E2 -1903.679} C_VEL
LIN {X 0,Y 580.601,Z 245.731,A -85,B 0,C 180,E1 -1906.707,E2 -1906.707} C_VEL
LIN {X 0,Y 580.807,Z 225.315,A -85,B 0,C 180,E1 -1909.294,E2 -1909.294} C_VEL
LIN {X 0,Y 581.011,Z 205.486,A -85,B 0,C 180,E1 -1911.836,E2 -1911.836} C_VEL
LIN {X 0,Y 580.969,Z 185.921,A -85,B 0,C 180,E1 -1914.286,E2 -1914.286} C_VEL
LIN {X 0,Y 580.264,Z 182.208,A -85,B 0,C 180,E1 -1914.793,E2 -1914.793} C_VEL
LIN {X 0,Y 580.258,Z 182.206,A -85,B 0,C 180,E1 -1917.403,E2 -1917.403} C_VEL
LIN {X 0,Y 580.254,Z 182.203,A -85,B 0,C 180,E1 -1919.774,E2 -1919.774} C_VEL
LIN {X 0,Y 580.284,Z 182.198,A -85,B 0,C 180,E1 -1922.201,E2 -1922.201} C_VEL
LIN {X 0,Y 580.283,Z 182.204,A -85,B 0,C 180,E1 -1924.697,E2 -1924.697} C_VEL
LIN {X 0,Y 580.286,Z 182.2,A -85,B 0,C 180,E1 -1927.269,E2 -1927.269} C_VEL
LIN {X 0,Y 580.282,Z 182.2,A -85,B 0,C 180,E1 -1930.269,E2 -1930.269} C_VEL
LIN {X 0,Y 580.272,Z 182.208,A -85,B 0,C 180,E1 -1932.707,E2 -1932.707} C_VEL
LIN {X 0,Y 580.255,Z 182.2,A -85,B 0,C 180,E1 -1935.61,E2 -1935.61} C_VEL
LIN {X 0,Y 580.273,Z 182.205,A -85,B 0,C 180,E1 -1938.67,E2 -1938.67} C_VEL
LIN {X 0,Y 580.269,Z 182.201,A -85,B 0,C 180,E1 -1940.964,E2 -1940.964} C_VEL
LIN {X 0,Y 580.248,Z 182.202,A -85,B 0,C 180,E1 -1943.595,E2 -1943.595} C_VEL
LIN {X 0,Y 580.3,Z 182.202,A -85,B 0,C 180,E1 -1946.144,E2 -1946.144} C_VEL
LIN {X 0,Y 580.267,Z 182.203,A -85,B 0,C 180,E1 -1948.614,E2 -1948.614} C_VEL
LIN {X 0,Y 580.285,Z 182.197,A -85,B 0,C 180,E1 -1951.023,E2 -1951.023} C_VEL
LIN {X 0,Y 580.267,Z 182.202,A -85,B 0,C 180,E1 -1953.671,E2 -1953.671} C_VEL
LIN {X 0,Y 580.262,Z 182.203,A -85,B 0,C 180,E1 -1956.441,E2 -1956.441} C_VEL
LIN {X 0,Y 580.268,Z 182.201,A -85,B 0,C 180,E1 -1959.437,E2 -1959.437} C_VEL
LIN {X 0,Y 580.25,Z 182.207,A -85,B 0,C 180,E1 -1961.644,E2 -1961.644} C_VEL
LIN {X 0,Y 580.257,Z 182.21,A -85,B 0,C 180,E1 -1963.825,E2 -1963.825} C_VEL
LIN {X 0,Y 580.313,Z 182.199,A -85,B 0,C 180,E1 -1965.983,E2 -1965.983} C_VEL
LIN {X 0,Y 580.306,Z 182.194,A -85,B 0,C 180,E1 -1968.827,E2 -1968.827} C_VEL
LIN {X 0,Y 580.327,Z 182.201,A -85,B 0,C 180,E1 -1971.644,E2 -1971.644} C_VEL
LIN {X 0,Y 580.32,Z 182.192,A -85,B 0,C 180,E1 -1974.44,E2 -1974.44} C_VEL
LIN {X 0,Y 580.347,Z 182.191,A -85,B 0,C 180,E1 -1977.918,E2 -1977.918} C_VEL
LIN {X 0,Y 580.35,Z 182.19,A -85,B 0,C 180,E1 -1980.694,E2 -1980.694} C_VEL
LIN {X 0,Y 580.286,Z 182.203,A -85,B 0,C 180,E1 -1983.472,E2 -1983.472} C_VEL
LIN {X 0,Y 580.333,Z 182.195,A -85,B 0,C 180,E1 -1985.56,E2 -1985.56} C_VEL
LIN {X 0,Y 580.31,Z 182.194,A -85,B 0,C 180,E1 -1988.356,E2 -1988.356} C_VEL
LIN {X 0,Y 580.301,Z 182.203,A -85,B 0,C 180,E1 -1991.191,E2 -1991.191} C_VEL
LIN {X 0,Y 580.326,Z 182.193,A -85,B 0,C 180,E1 -1994.017,E2 -1994.017} C_VEL
LIN {X 0,Y 580.313,Z 182.203,A -85,B 0,C 180,E1 -1996.914,E2 -1996.914} C_VEL
LIN {X 0,Y 580.286,Z 182.197,A -85,B 0,C 180,E1 -1999.823,E2 -1999.823} C_VEL
LIN {X 0,Y 580.29,Z 182.2,A -85,B 0,C 180,E1 -2001.311,E2 -2001.311} C_VEL
LIN {X 0,Y 579.94,Z 182.499,A -85,B 0,C 180,E1 -2001.695,E2 -2001.695} C_VEL
LIN {X 0,Y 578.54,Z 183.842,A -85,B 0,C 180,E1 -2002.247,E2 -2002.247} C_VEL
LIN {X 0,Y 576.641,Z 185.922,A -85,B 0,C 180,E1 -2002.769,E2 -2002.769} C_VEL
LIN {X 0,Y 573.782,Z 190.411,A -85,B 0,C 180,E1 -2003.632,E2 -2003.632} C_VEL
LIN {X 0,Y 573.215,Z 193.051,A -85,B 0,C 180,E1 -2004.168,E2 -2004.168} C_VEL
LIN {X 0,Y 573.221,Z 193.332,A -85,B 0,C 180,E1 -2004.227,E2 -2004.227} C_VEL
LIN {X 0,Y 574.069,Z 198.998,A -85,B 0,C 180,E1 -2004.333,E2 -2004.333} C_VEL
LIN {X 0,Y 573.863,Z 299.452,A -85,B 0,C 180,E1 -2005.612,E2 -2005.612} C_VEL
LIN {X 0,Y 573.767,Z 312.442,A -85,B 0,C 180,E1 -2005.921,E2 -2005.921} C_VEL
LIN {X 0,Y 573.688,Z 324.761,A -85,B 0,C 180,E1 -2006.354,E2 -2006.354} C_VEL
LIN {X 0,Y 573.57,Z 336.34,A -85,B 0,C 180,E1 -2006.902,E2 -2006.902} C_VEL
LIN {X 0,Y 573.445,Z 347.162,A -85,B 0,C 180,E1 -2007.559,E2 -2007.559} C_VEL
LIN {X 0,Y 573.323,Z 358.407,A -85,B 0,C 180,E1 -2008.414,E2 -2008.414} C_VEL
LIN {X 0,Y 573.234,Z 366.482,A -85,B 0,C 180,E1 -2009.166,E2 -2009.166} C_VEL
LIN {X 0,Y 573.162,Z 375.474,A -85,B 0,C 180,E1 -2010.181,E2 -2010.181} C_VEL
LIN {X 0,Y 573.078,Z 382.809,A -85,B 0,C 180,E1 -2011.207,E2 -2011.207} C_VEL
LIN {X 0,Y 573.04,Z 389.614,A -85,B 0,C 180,E1 -2012.402,E2 -2012.402} C_VEL
LIN {X 0,Y 572.992,Z 394.486,A -85,B 0,C 180,E1 -2013.501,E2 -2013.501} C_VEL
LIN {X 0,Y 572.988,Z 398.558,A -85,B 0,C 180,E1 -2014.736,E2 -2014.736} C_VEL
LIN {X 0,Y 572.923,Z 401.417,A -85,B 0,C 180,E1 -2016.073,E2 -2016.073} C_VEL
LIN {X 0,Y 572.926,Z 402.638,A -85,B 0,C 180,E1 -2017.123,E2 -2017.123} C_VEL
LIN {X 0,Y 572.929,Z 402.956,A -85,B 0,C 180,E1 -2018.273,E2 -2018.273} C_VEL
LIN {X 0,Y 572.927,Z 401.976,A -85,B 0,C 180,E1 -2019.634,E2 -2019.634} C_VEL
LIN {X 0,Y 572.938,Z 399.414,A -85,B 0,C 180,E1 -2021.016,E2 -2021.016} C_VEL
LIN {X 0,Y 573.007,Z 396.726,A -85,B 0,C 180,E1 -2021.966,E2 -2021.966} C_VEL
LIN {X 0,Y 573.021,Z 392.946,A -85,B 0,C 180,E1 -2022.971,E2 -2022.971} C_VEL
LIN {X 0,Y 573.061,Z 387.135,A -85,B 0,C 180,E1 -2024.16,E2 -2024.16} C_VEL
LIN {X 0,Y 573.096,Z 379.735,A -85,B 0,C 180,E1 -2025.338,E2 -2025.338} C_VEL
LIN {X 0,Y 573.177,Z 371.91,A -85,B 0,C 180,E1 -2026.338,E2 -2026.338} C_VEL
LIN {X 0,Y 573.274,Z 363.453,A -85,B 0,C 180,E1 -2027.224,E2 -2027.224} C_VEL
LIN {X 0,Y 573.389,Z 352.665,A -85,B 0,C 180,E1 -2028.137,E2 -2028.137} C_VEL
LIN {X 0,Y 573.473,Z 341.236,A -85,B 0,C 180,E1 -2028.911,E2 -2028.911} C_VEL
LIN {X 0,Y 573.627,Z 329.959,A -85,B 0,C 180,E1 -2029.508,E2 -2029.508} C_VEL
LIN {X 0,Y 573.771,Z 316.647,A -85,B 0,C 180,E1 -2030.037,E2 -2030.037} C_VEL
LIN {X 0,Y 573.863,Z 304.035,A -85,B 0,C 180,E1 -2030.387,E2 -2030.387} C_VEL
LIN {X 0,Y 573.915,Z 289.52,A -85,B 0,C 180,E1 -2030.622,E2 -2030.622} C_VEL
LIN {X 0,Y 574.066,Z 198.31,A -85,B 0,C 180,E1 -2031.766,E2 -2031.766} C_VEL
LIN {X 0,Y 573.171,Z 193.346,A -85,B 0,C 180,E1 -2031.862,E2 -2031.862} C_VEL
LIN {X 0,Y 573.261,Z 183.075,A -85,B 0,C 180,E1 -2034.012,E2 -2034.012} C_VEL
LIN {X 0,Y 573.233,Z 183.077,A -85,B 0,C 180,E1 -2036.516,E2 -2036.516} C_VEL
LIN {X 0,Y 573.222,Z 183.085,A -85,B 0,C 180,E1 -2039.119,E2 -2039.119} C_VEL
LIN {X 0,Y 573.234,Z 183.081,A -85,B 0,C 180,E1 -2041.436,E2 -2041.436} C_VEL
LIN {X 0,Y 573.234,Z 183.077,A -85,B 0,C 180,E1 -2044.589,E2 -2044.589} C_VEL
LIN {X 0,Y 573.222,Z 183.078,A -85,B 0,C 180,E1 -2047.662,E2 -2047.662} C_VEL
LIN {X 0,Y 573.237,Z 183.074,A -85,B 0,C 180,E1 -2049.923,E2 -2049.923} C_VEL
LIN {X 0,Y 573.238,Z 183.083,A -85,B 0,C 180,E1 -2052.998,E2 -2052.998} C_VEL
LIN {X 0,Y 573.253,Z 183.072,A -85,B 0,C 180,E1 -2055.807,E2 -2055.807} C_VEL
LIN {X 0,Y 573.265,Z 183.081,A -85,B 0,C 180,E1 -2058.745,E2 -2058.745} C_VEL
LIN {X 0,Y 573.252,Z 183.073,A -85,B 0,C 180,E1 -2061.54,E2 -2061.54} C_VEL
LIN {X 0,Y 573.296,Z 183.073,A -85,B 0,C 180,E1 -2064.372,E2 -2064.372} C_VEL
LIN {X 0,Y 573.312,Z 183.066,A -85,B 0,C 180,E1 -2067.893,E2 -2067.893} C_VEL
LIN {X 0,Y 573.329,Z 183.069,A -85,B 0,C 180,E1 -2070.703,E2 -2070.703} C_VEL
LIN {X 0,Y 573.294,Z 183.071,A -85,B 0,C 180,E1 -2072.811,E2 -2072.811} C_VEL
LIN {X 0,Y 573.283,Z 183.069,A -85,B 0,C 180,E1 -2075.628,E2 -2075.628} C_VEL
LIN {X 0,Y 573.281,Z 183.076,A -85,B 0,C 180,E1 -2078.46,E2 -2078.46} C_VEL
LIN {X 0,Y 573.275,Z 183.07,A -85,B 0,C 180,E1 -2081.312,E2 -2081.312} C_VEL
LIN {X 0,Y 573.27,Z 183.076,A -85,B 0,C 180,E1 -2084.419,E2 -2084.419} C_VEL
LIN {X 0,Y 573.248,Z 183.073,A -85,B 0,C 180,E1 -2087.112,E2 -2087.112} C_VEL
LIN {X 0,Y 573.237,Z 183.084,A -85,B 0,C 180,E1 -2090.077,E2 -2090.077} C_VEL
LIN {X 0,Y 573.223,Z 183.08,A -85,B 0,C 180,E1 -2092.339,E2 -2092.339} C_VEL
LIN {X 0,Y 573.237,Z 183.077,A -85,B 0,C 180,E1 -2095.411,E2 -2095.411} C_VEL
LIN {X 0,Y 573.223,Z 183.077,A -85,B 0,C 180,E1 -2098.566,E2 -2098.566} C_VEL
LIN {X 0,Y 573.22,Z 183.077,A -85,B 0,C 180,E1 -2100.994,E2 -2100.994} C_VEL
LIN {X 0,Y 573.266,Z 183.078,A -85,B 0,C 180,E1 -2103.524,E2 -2103.524} C_VEL
LIN {X 0,Y 573.194,Z 183.083,A -85,B 0,C 180,E1 -2106.053,E2 -2106.053} C_VEL
LIN {X 0,Y 573.237,Z 183.075,A -85,B 0,C 180,E1 -2108.702,E2 -2108.702} C_VEL
LIN {X 0,Y 573.224,Z 183.085,A -85,B 0,C 180,E1 -2111.592,E2 -2111.592} C_VEL
LIN {X 0,Y 573.224,Z 183.076,A -85,B 0,C 180,E1 -2114.335,E2 -2114.335} C_VEL
LIN {X 0,Y 573.239,Z 183.084,A -85,B 0,C 180,E1 -2117.359,E2 -2117.359} C_VEL
LIN {X 0,Y 573.235,Z 183.075,A -85,B 0,C 180,E1 -2120.392,E2 -2120.392} C_VEL
LIN {X 0,Y 573.234,Z 183.082,A -85,B 0,C 180,E1 -2123.076,E2 -2123.076} C_VEL
LIN {X 0,Y 573.255,Z 183.075,A -85,B 0,C 180,E1 -2125.67,E2 -2125.67} C_VEL
LIN {X 0,Y 573.228,Z 183.076,A -85,B 0,C 180,E1 -2128.184,E2 -2128.184} C_VEL
LIN {X 0,Y 573.241,Z 183.077,A -85,B 0,C 180,E1 -2130.633,E2 -2130.633} C_VEL
LIN {X 0,Y 573.234,Z 183.077,A -85,B 0,C 180,E1 -2133.509,E2 -2133.509} C_VEL
LIN {X 0,Y 573.201,Z 183.079,A -85,B 0,C 180,E1 -2136.133,E2 -2136.133} C_VEL
LIN {X 0,Y 573.255,Z 183.08,A -85,B 0,C 180,E1 -2138.71,E2 -2138.71} C_VEL
LIN {X 0,Y 573.203,Z 183.08,A -85,B 0,C 180,E1 -2141.411,E2 -2141.411} C_VEL
LIN {X 0,Y 573.228,Z 183.076,A -85,B 0,C 180,E1 -2143.621,E2 -2143.621} C_VEL
LIN {X 0,Y 573.244,Z 183.074,A -85,B 0,C 180,E1 -2145.806,E2 -2145.806} C_VEL
LIN {X 0,Y 573.267,Z 183.079,A -85,B 0,C 180,E1 -2148.745,E2 -2148.745} C_VEL
LIN {X 0,Y 573.248,Z 183.073,A -85,B 0,C 180,E1 -2151.54,E2 -2151.54} C_VEL
LIN {X 0,Y 573.282,Z 183.077,A -85,B 0,C 180,E1 -2154.372,E2 -2154.372} C_VEL
LIN {X 0,Y 573.311,Z 183.068,A -85,B 0,C 180,E1 -2157.892,E2 -2157.892} C_VEL
LIN {X 0,Y 573.322,Z 183.068,A -85,B 0,C 180,E1 -2160.702,E2 -2160.702} C_VEL
LIN {X 0,Y 573.286,Z 183.071,A -85,B 0,C 180,E1 -2162.811,E2 -2162.811} C_VEL
LIN {X 0,Y 573.28,Z 183.071,A -85,B 0,C 180,E1 -2165.628,E2 -2165.628} C_VEL
LIN {X 0,Y 573.25,Z 183.078,A -85,B 0,C 180,E1 -2168.46,E2 -2168.46} C_VEL
LIN {X 0,Y 573.276,Z 183.07,A -85,B 0,C 180,E1 -2171.312,E2 -2171.312} C_VEL
LIN {X 0,Y 573.274,Z 183.074,A -85,B 0,C 180,E1 -2174.42,E2 -2174.42} C_VEL
LIN {X 0,Y 573.197,Z 183.08,A -85,B 0,C 180,E1 -2177.114,E2 -2177.114} C_VEL
LIN {X 0,Y 573.269,Z 183.072,A -85,B 0,C 180,E1 -2179.33,E2 -2179.33} C_VEL
LIN {X 0,Y 573.222,Z 183.079,A -85,B 0,C 180,E1 -2182.339,E2 -2182.339} C_VEL
LIN {X 0,Y 573.233,Z 183.079,A -85,B 0,C 180,E1 -2185.411,E2 -2185.411} C_VEL
LIN {X 0,Y 573.202,Z 183.079,A -85,B 0,C 180,E1 -2188.567,E2 -2188.567} C_VEL
LIN {X 0,Y 573.219,Z 183.078,A -85,B 0,C 180,E1 -2190.994,E2 -2190.994} C_VEL
LIN {X 0,Y 573.245,Z 183.083,A -85,B 0,C 180,E1 -2193.521,E2 -2193.521} C_VEL
LIN {X 0,Y 573.19,Z 183.082,A -85,B 0,C 180,E1 -2196.053,E2 -2196.053} C_VEL
LIN {X 0,Y 573.235,Z 183.075,A -85,B 0,C 180,E1 -2198.702,E2 -2198.702} C_VEL
LIN {X 0,Y 573.212,Z 183.084,A -85,B 0,C 180,E1 -2201.59,E2 -2201.59} C_VEL
LIN {X 0,Y 573.21,Z 183.079,A -85,B 0,C 180,E1 -2204.673,E2 -2204.673} C_VEL
LIN {X 0,Y 573.214,Z 183.081,A -85,B 0,C 180,E1 -2207.597,E2 -2207.597} C_VEL
LIN {X 0,Y 573.236,Z 183.076,A -85,B 0,C 180,E1 -2210.57,E2 -2210.57} C_VEL
LIN {X 0,Y 573.233,Z 183.085,A -85,B 0,C 180,E1 -2213.076,E2 -2213.076} C_VEL
LIN {X 0,Y 573.249,Z 183.074,A -85,B 0,C 180,E1 -2215.67,E2 -2215.67} C_VEL
LIN {X 0,Y 573.227,Z 183.077,A -85,B 0,C 180,E1 -2218.183,E2 -2218.183} C_VEL
LIN {X 0,Y 573.234,Z 183.081,A -85,B 0,C 180,E1 -2220.632,E2 -2220.632} C_VEL
LIN {X 0,Y 573.215,Z 183.08,A -85,B 0,C 180,E1 -2223.513,E2 -2223.513} C_VEL
LIN {X 0,Y 573.238,Z 183.124,A -85,B 0,C 180,E1 -2225.015,E2 -2225.015} C_VEL
LIN {X 0,Y 574.157,Z 188.757,A -85,B 0,C 180,E1 -2225.791,E2 -2225.791} C_VEL
LIN {X 0,Y 574.008,Z 209.99,A -85,B 0,C 180,E1 -2228.517,E2 -2228.517} C_VEL
LIN {X 0,Y 573.834,Z 229.942,A -85,B 0,C 180,E1 -2231.061,E2 -2231.061} C_VEL
LIN {X 0,Y 573.61,Z 252.903,A -85,B 0,C 180,E1 -2233.998,E2 -2233.998} C_VEL
LIN {X 0,Y 573.473,Z 270.229,A -85,B 0,C 180,E1 -2236.162,E2 -2236.162} C_VEL
LIN {X 0,Y 574.053,Z 276.49,A -85,B 0,C 180,E1 -2236.256,E2 -2236.256} C_VEL
LIN {X 0,Y 573.908,Z 378.935,A -85,B 0,C 180,E1 -2237.558,E2 -2237.558} C_VEL
LIN {X 0,Y 573.776,Z 392.211,A -85,B 0,C 180,E1 -2237.869,E2 -2237.869} C_VEL
LIN {X 0,Y 573.678,Z 405.148,A -85,B 0,C 180,E1 -2238.324,E2 -2238.324} C_VEL
LIN {X 0,Y 573.586,Z 416.669,A -85,B 0,C 180,E1 -2238.876,E2 -2238.876} C_VEL
LIN {X 0,Y 573.428,Z 428.196,A -85,B 0,C 180,E1 -2239.585,E2 -2239.585} C_VEL
LIN {X 0,Y 573.333,Z 438.599,A -85,B 0,C 180,E1 -2240.385,E2 -2240.385} C_VEL
LIN {X 0,Y 573.241,Z 447.111,A -85,B 0,C 180,E1 -2241.184,E2 -2241.184} C_VEL
LIN {X 0,Y 573.161,Z 454.959,A -85,B 0,C 180,E1 -2242.071,E2 -2242.071} C_VEL
LIN {X 0,Y 573.073,Z 462.954,A -85,B 0,C 180,E1 -2243.185,E2 -2243.185} C_VEL
LIN {X 0,Y 573.07,Z 469.679,A -85,B 0,C 180,E1 -2244.369,E2 -2244.369} C_VEL
LIN {X 0,Y 573.028,Z 474.371,A -85,B 0,C 180,E1 -2245.427,E2 -2245.427} C_VEL
LIN {X 0,Y 573.022,Z 477.957,A -85,B 0,C 180,E1 -2246.484,E2 -2246.484} C_VEL
LIN {X 0,Y 572.959,Z 479.807,A -85,B 0,C 180,E1 -2247.187,E2 -2247.187} C_VEL
LIN {X 0,Y 572.94,Z 481.197,A -85,B 0,C 180,E1 -2247.891,E2 -2247.891} C_VEL
LIN {X 0,Y 572.94,Z 482.785,A -85,B 0,C 180,E1 -2249.297,E2 -2249.297} C_VEL
LIN {X 0,Y 572.938,Z 483,A -85,B 0,C 180,E1 -2250,E2 -2250} C_VEL
LIN {X 0,Y 572.946,Z 482.186,A -85,B 0,C 180,E1 -2251.406,E2 -2251.406} C_VEL
LIN {X 0,Y 572.94,Z 481.199,A -85,B 0,C 180,E1 -2252.109,E2 -2252.109} C_VEL
LIN {X 0,Y 572.959,Z 479.81,A -85,B 0,C 180,E1 -2252.812,E2 -2252.812} C_VEL
LIN {X 0,Y 573.015,Z 476.896,A -85,B 0,C 180,E1 -2253.868,E2 -2253.868} C_VEL
LIN {X 0,Y 572.963,Z 472.95,A -85,B 0,C 180,E1 -2254.925,E2 -2254.925} C_VEL
LIN {X 0,Y 573.065,Z 466.878,A -85,B 0,C 180,E1 -2256.16,E2 -2256.16} C_VEL
LIN {X 0,Y 573.119,Z 460.238,A -85,B 0,C 180,E1 -2257.221,E2 -2257.221} C_VEL
LIN {X 0,Y 573.201,Z 451.992,A -85,B 0,C 180,E1 -2258.283,E2 -2258.283} C_VEL
LIN {X 0,Y 573.287,Z 443.541,A -85,B 0,C 180,E1 -2259.17,E2 -2259.17} C_VEL
LIN {X 0,Y 573.427,Z 433.099,A -85,B 0,C 180,E1 -2260.058,E2 -2260.058} C_VEL
LIN {X 0,Y 573.543,Z 421.435,A -85,B 0,C 180,E1 -2260.853,E2 -2260.853} C_VEL
LIN {X 0,Y 573.651,Z 410.309,A -85,B 0,C 180,E1 -2261.446,E2 -2261.446} C_VEL
LIN {X 0,Y 573.756,Z 397.175,A -85,B 0,C 180,E1 -2261.974,E2 -2261.974} C_VEL
LIN {X 0,Y 573.849,Z 384.524,A -85,B 0,C 180,E1 -2262.331,E2 -2262.331} C_VEL
LIN {X 0,Y 573.933,Z 371.322,A -85,B 0,C 180,E1 -2262.554,E2 -2262.554} C_VEL
LIN {X 0,Y 573.967,Z 273.615,A -85,B 0,C 180,E1 -2263.783,E2 -2263.783} C_VEL
LIN {X 0,Y 573.465,Z 269.947,A -85,B 0,C 180,E1 -2263.849,E2 -2263.849} C_VEL
LIN {X 0,Y 573.636,Z 245.741,A -85,B 0,C 180,E1 -2266.915,E2 -2266.915} C_VEL
LIN {X 0,Y 573.872,Z 226.067,A -85,B 0,C 180,E1 -2269.439,E2 -2269.439} C_VEL
LIN {X 0,Y 574.028,Z 204.785,A -85,B 0,C 180,E1 -2272.116,E2 -2272.116} C_VEL
LIN {X 0,Y 574.054,Z 188.227,A -85,B 0,C 180,E1 -2274.213,E2 -2274.213} C_VEL
LIN {X 0,Y 573.223,Z 183.086,A -85,B 0,C 180,E1 -2274.912,E2 -2274.912} C_VEL
LIN {X 0,Y 573.227,Z 183.079,A -85,B 0,C 180,E1 -2277.768,E2 -2277.768} C_VEL
LIN {X 0,Y 573.22,Z 183.079,A -85,B 0,C 180,E1 -2280.178,E2 -2280.178} C_VEL
LIN {X 0,Y 573.246,Z 183.079,A -85,B 0,C 180,E1 -2282.645,E2 -2282.645} C_VEL
LIN {X 0,Y 573.202,Z 183.084,A -85,B 0,C 180,E1 -2285.188,E2 -2285.188} C_VEL
LIN {X 0,Y 573.227,Z 183.076,A -85,B 0,C 180,E1 -2287.808,E2 -2287.808} C_VEL
LIN {X 0,Y 573.246,Z 183.08,A -85,B 0,C 180,E1 -2290.525,E2 -2290.525} C_VEL
LIN {X 0,Y 573.208,Z 183.079,A -85,B 0,C 180,E1 -2293.362,E2 -2293.362} C_VEL
LIN {X 0,Y 573.236,Z 183.081,A -85,B 0,C 180,E1 -2296.332,E2 -2296.332} C_VEL
